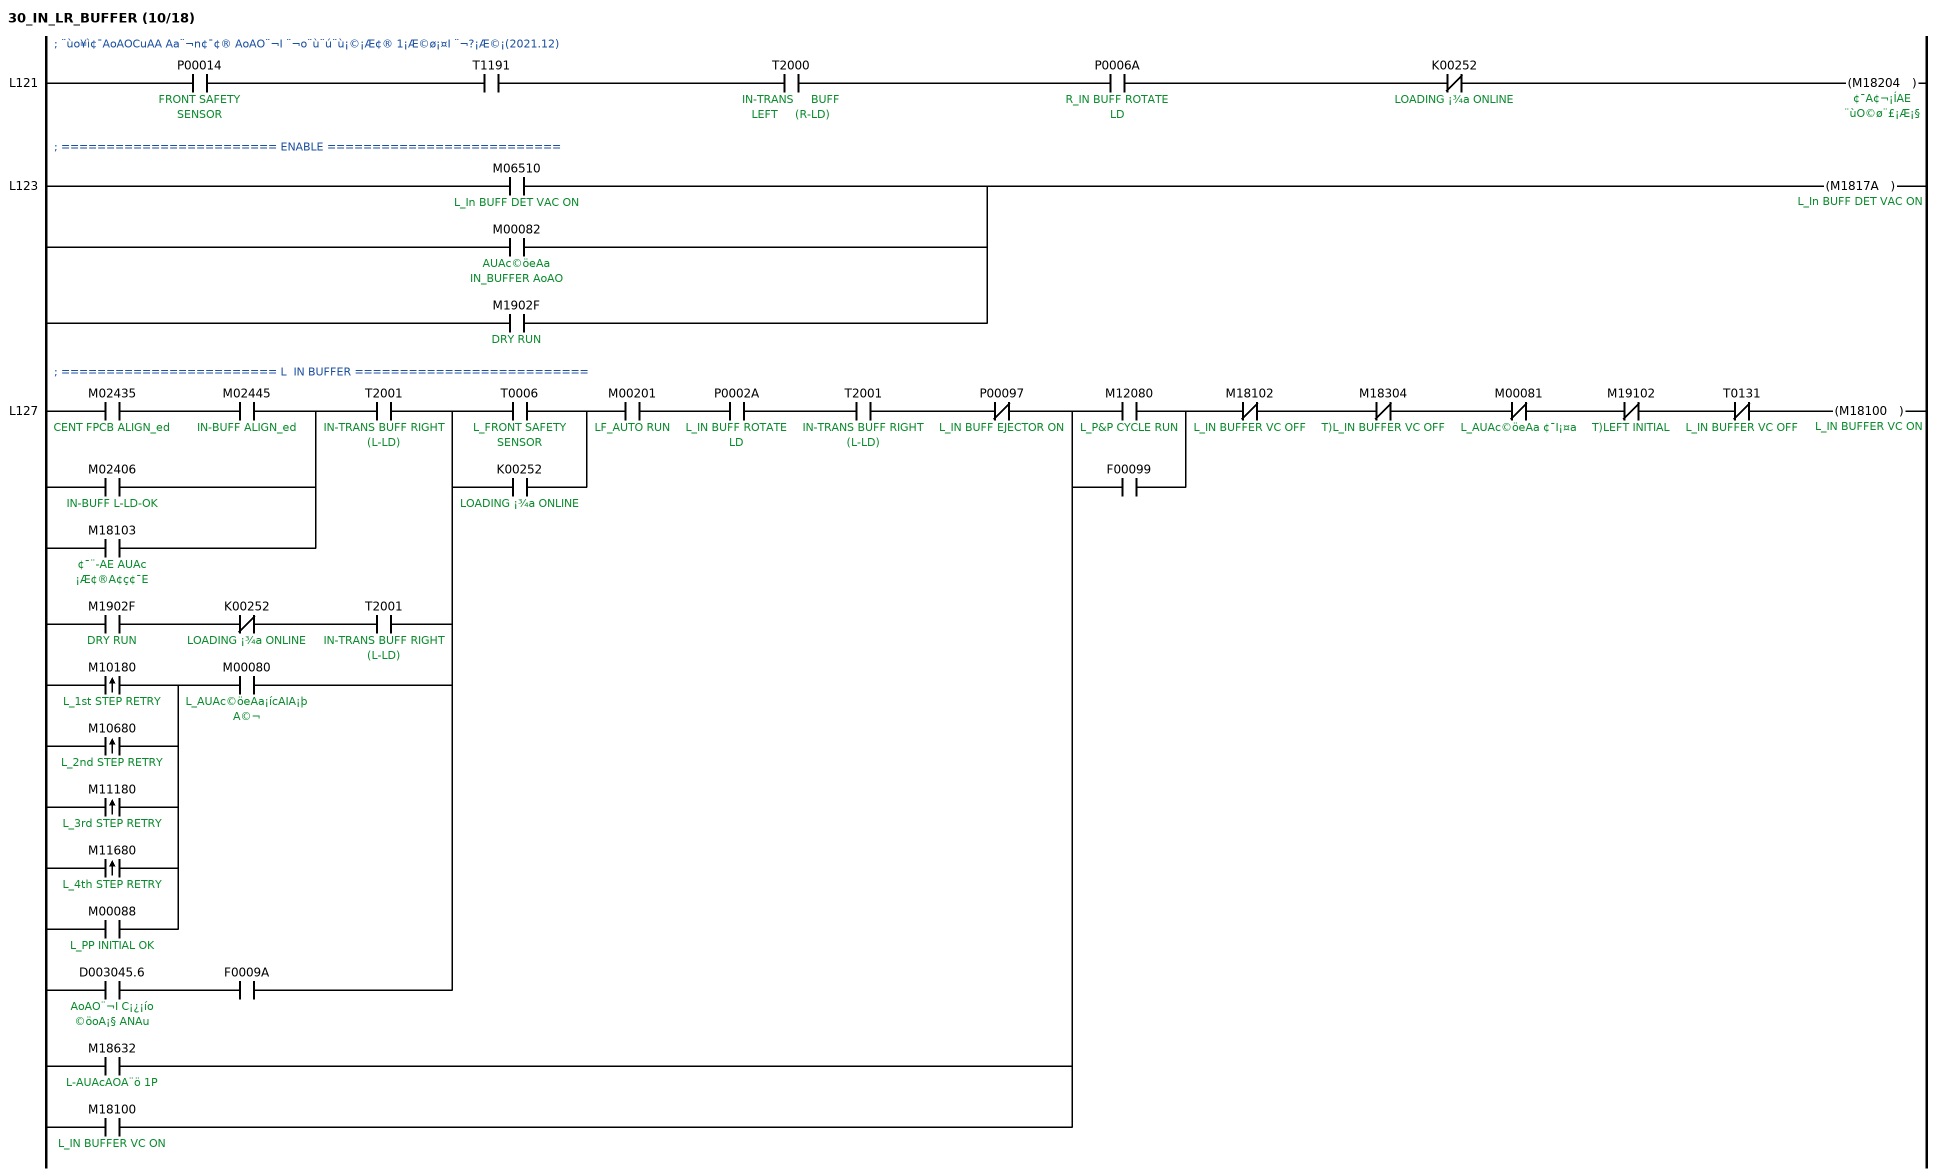
[picture p216: 30_IN_LR_BUFFER rungs L121-L127]
; L121
LOAD      P00014	// FRONT SAFETY SENSOR
AND       T1191
AND       T2000	// IN-TRANS     BUFF     LEFT     (R-LD)
AND       P0006A	// R_IN BUFF ROTATE      LD
AND NOT   K00252	// LOADING ¡¾a ONLINE
OUT       M18204	// ¢¯A¢¬¡ÍAE ¨ùO©ø¨£¡Æ¡§
// output comment: ¨ùo¥ì¢¯AoAOCuAA Aa¨¬n¢¯¢® AoAO¨¬I ¨¬o¨ù¨ú¨ù¡©¡Æ¢® 1¡Æ©ø¡¤I ¨¬?¡Æ©¡(2021.12)
// ======================== ENABLE ==========================
; L123
LOAD      M06510	// L_In BUFF DET VAC ON
OR        M00082	// AUAc©öeAa IN_BUFFER AoAO 
OR        M1902F	// DRY RUN
OUT       M1817A	// L_In BUFF DET VAC ON
// ======================== L  IN BUFFER ==========================
; L127
LOAD      M02435	// CENT FPCB ALIGN_ed
AND       M02445	// IN-BUFF ALIGN_ed
OR        M02406	// IN-BUFF L-LD-OK
OR        M18103	// ¢¯¨­AE AUAc ¡Æ¢®A¢ç¢¯E
AND       T2001	// IN-TRANS BUFF RIGHT     (L-LD)
LOAD      M1902F	// DRY RUN
AND NOT   K00252	// LOADING ¡¾a ONLINE
AND       T2001	// IN-TRANS BUFF RIGHT     (L-LD)
OR LOAD
LOADP     M10180	// L_1st STEP RETRY
ORP       M10680	// L_2nd STEP RETRY
ORP       M11180	// L_3rd STEP RETRY
ORP       M11680	// L_4th STEP RETRY
OR        M00088	// L_PP INITIAL OK
AND       M00080	// L_AUAc©öeAa¡ícAIA¡þA©¬
OR LOAD
LOAD      D003045.6	// AoAO¨¬I C¡¿¡ío ©öoA¡§ ANAu
AND       F0009A
OR LOAD
LOAD      T0006	// L_FRONT SAFETY SENSOR
OR        K00252	// LOADING ¡¾a ONLINE
AND LOAD
AND       M00201	// LF_AUTO RUN
AND       P0002A	// L_IN BUFF ROTATE     LD
AND       T2001	// IN-TRANS BUFF RIGHT     (L-LD)
AND NOT   P00097	// L_IN BUFF EJECTOR ON
OR        M18632	// L-AUAcAOA¨ö 1P
OR        M18100	// L_IN BUFFER VC ON
LOAD      M12080	// L_P&P CYCLE RUN
OR        F00099
AND LOAD
AND NOT   M18102	// L_IN BUFFER VC OFF
AND NOT   M18304	// T)L_IN BUFFER VC OFF
AND NOT   M00081	// L_AUAc©öeAa ¢¯I¡¤a
AND NOT   M19102	// T)LEFT INITIAL
AND NOT   T0131	// L_IN BUFFER VC OFF
OUT       M18100	// L_IN BUFFER VC ON

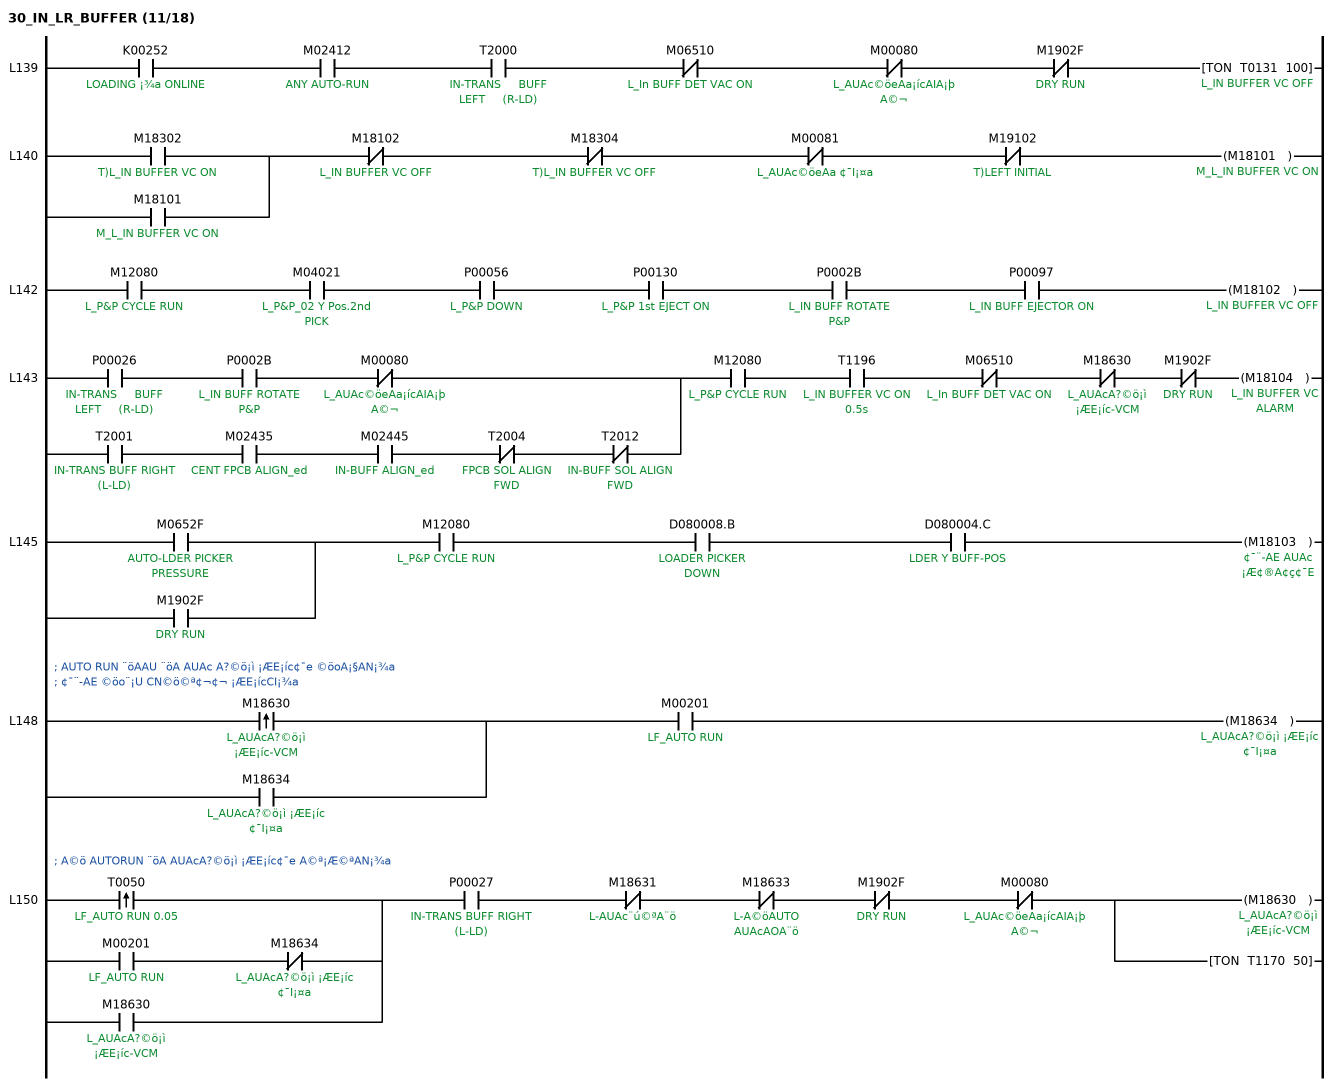
; L139
LOAD      K00252	// LOADING ¡¾a ONLINE
AND       M02412	// ANY AUTO-RUN
AND       T2000	// IN-TRANS     BUFF     LEFT     (R-LD)
AND NOT   M06510	// L_In BUFF DET VAC ON
AND NOT   M00080	// L_AUAc©öeAa¡ícAIA¡þA©¬
AND NOT   M1902F	// DRY RUN
TON       T0131 100	// L_IN BUFFER VC OFF
; L140
LOAD      M18302	// T)L_IN BUFFER VC ON
OR        M18101	// M_L_IN BUFFER VC ON
AND NOT   M18102	// L_IN BUFFER VC OFF
AND NOT   M18304	// T)L_IN BUFFER VC OFF
AND NOT   M00081	// L_AUAc©öeAa ¢¯I¡¤a
AND NOT   M19102	// T)LEFT INITIAL
OUT       M18101	// M_L_IN BUFFER VC ON
; L142
LOAD      M12080	// L_P&P CYCLE RUN
AND       M04021	// L_P&P_02 Y Pos.2nd PICK
AND       P00056	// L_P&P DOWN
AND       P00130	// L_P&P 1st EJECT ON
AND       P0002B	// L_IN BUFF ROTATE      P&P
AND       P00097	// L_IN BUFF EJECTOR ON
OUT       M18102	// L_IN BUFFER VC OFF
; L143
LOAD      P00026	// IN-TRANS     BUFF     LEFT     (R-LD)
AND       P0002B	// L_IN BUFF ROTATE      P&P
AND NOT   M00080	// L_AUAc©öeAa¡ícAIA¡þA©¬
LOAD      T2001	// IN-TRANS BUFF RIGHT     (L-LD)
AND       M02435	// CENT FPCB ALIGN_ed
AND       M02445	// IN-BUFF ALIGN_ed
AND NOT   T2004	// FPCB SOL ALIGN         FWD
AND NOT   T2012	// IN-BUFF SOL ALIGN FWD
OR LOAD
AND       M12080	// L_P&P CYCLE RUN
AND       T1196	// L_IN BUFFER VC ON 0.5s
AND NOT   M06510	// L_In BUFF DET VAC ON
AND NOT   M18630	// L_AUAcA?©ö¡ì ¡ÆE¡íc-VCM
AND NOT   M1902F	// DRY RUN
OUT       M18104	// L_IN BUFFER VC ALARM
; L145
LOAD      M0652F	// AUTO-LDER PICKER PRESSURE
OR        M1902F	// DRY RUN
AND       M12080	// L_P&P CYCLE RUN
AND       D080008.B	// LOADER PICKER DOWN
AND       D080004.C	// LDER Y BUFF-POS
OUT       M18103	// ¢¯¨­AE AUAc ¡Æ¢®A¢ç¢¯E
// AUTO RUN ¨öAAU ¨öA AUAc A?©ö¡ì ¡ÆE¡íc¢¯e ©öoA¡§AN¡¾a
; L148
LOADP     M18630	// L_AUAcA?©ö¡ì ¡ÆE¡íc-VCM
OR        M18634	// L_AUAcA?©ö¡ì ¡ÆE¡íc ¢¯I¡¤a
AND       M00201	// LF_AUTO RUN
OUT       M18634	// L_AUAcA?©ö¡ì ¡ÆE¡íc ¢¯I¡¤a
// output comment: ¢¯¨­AE ©öo¨¡U CN©ö©ª¢¬¢¬ ¡ÆE¡ícCI¡¾a
; L150
LOADP     T0050	// LF_AUTO RUN 0.05
LOAD      M00201	// LF_AUTO RUN
AND NOT   M18634	// L_AUAcA?©ö¡ì ¡ÆE¡íc ¢¯I¡¤a
OR LOAD
OR        M18630	// L_AUAcA?©ö¡ì ¡ÆE¡íc-VCM
AND       P00027	// IN-TRANS BUFF RIGHT     (L-LD)
AND NOT   M18631	// L-AUAc¨ú©ªA¨ö
AND NOT   M18633	// L-A©öAUTO AUAcAOA¨ö
AND NOT   M1902F	// DRY RUN
AND NOT   M00080	// L_AUAc©öeAa¡ícAIA¡þA©¬
OUT       M18630	// L_AUAcA?©ö¡ì ¡ÆE¡íc-VCM
TON       T1170 50
// output comment: A©ö AUTORUN ¨öA AUAcA?©ö¡ì ¡ÆE¡íc¢¯e A©ª¡Æ©ªAN¡¾a

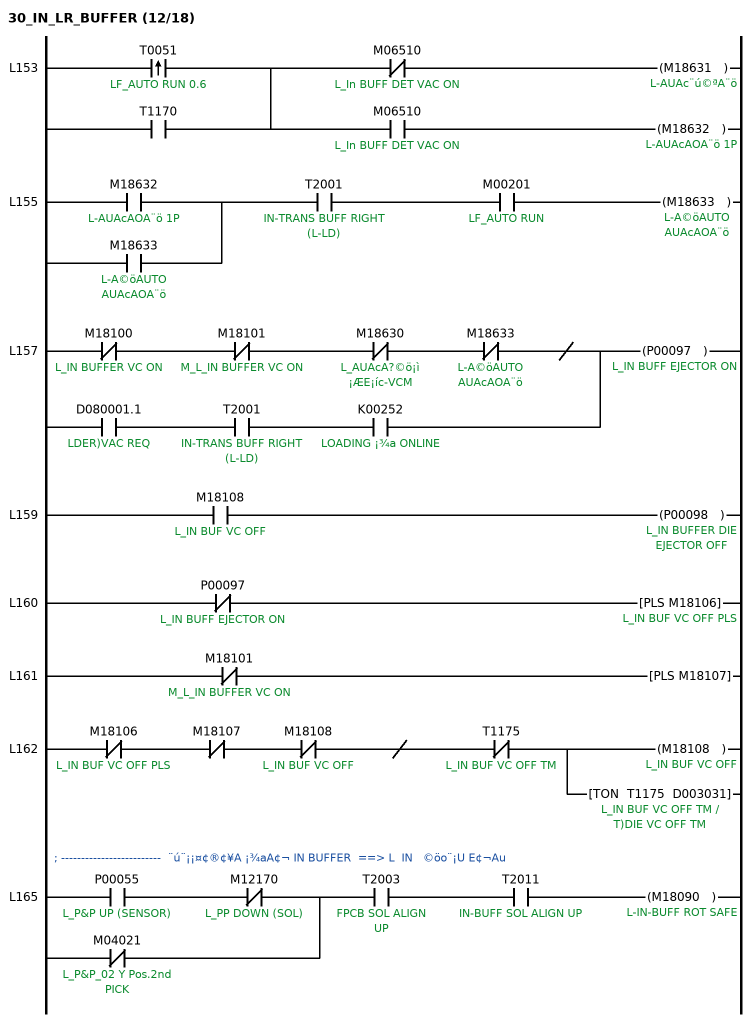
; L153
LOADP     T0051	// LF_AUTO RUN 0.6
OR        T1170
MPUSH
AND NOT   M06510	// L_In BUFF DET VAC ON
OUT       M18631	// L-AUAc¨ú©ªA¨ö
MPOP
AND       M06510	// L_In BUFF DET VAC ON
OUT       M18632	// L-AUAcAOA¨ö 1P
; L155
LOAD      M18632	// L-AUAcAOA¨ö 1P
OR        M18633	// L-A©öAUTO AUAcAOA¨ö
AND       T2001	// IN-TRANS BUFF RIGHT     (L-LD)
AND       M00201	// LF_AUTO RUN
OUT       M18633	// L-A©öAUTO AUAcAOA¨ö
; L157
LOAD NOT  M18100	// L_IN BUFFER VC ON
AND NOT   M18101	// M_L_IN BUFFER VC ON
AND NOT   M18630	// L_AUAcA?©ö¡ì ¡ÆE¡íc-VCM
AND NOT   M18633	// L-A©öAUTO AUAcAOA¨ö
NOT
LOAD      D080001.1	// LDER)VAC REQ
AND       T2001	// IN-TRANS BUFF RIGHT     (L-LD)
AND       K00252	// LOADING ¡¾a ONLINE
OR LOAD
OUT       P00097	// L_IN BUFF EJECTOR ON
; L159
LOAD      M18108	// L_IN BUF VC OFF
OUT       P00098	// L_IN BUFFER DIE EJECTOR OFF
; L160
LOAD NOT  P00097	// L_IN BUFF EJECTOR ON
OUTP      M18106	// L_IN BUF VC OFF PLS
; L161
LOAD NOT  M18101	// M_L_IN BUFFER VC ON
OUTP      M18107
; L162
LOAD NOT  M18106	// L_IN BUF VC OFF PLS
AND NOT   M18107
AND NOT   M18108	// L_IN BUF VC OFF
NOT
AND NOT   T1175	// L_IN BUF VC OFF TM
OUT       M18108	// L_IN BUF VC OFF
TON       T1175 D003031	// L_IN BUF VC OFF TM / T)DIE VC OFF TM
// -------------------------  ¨ú¨¡¡¤¢®¢¥A ¡¾aA¢¬ IN BUFFER  ==> L  IN   ©öo¨¡U E¢¬Au
; L165
LOAD      P00055	// L_P&P UP (SENSOR)
AND NOT   M12170	// L_PP DOWN (SOL)
OR NOT    M04021	// L_P&P_02 Y Pos.2nd PICK
AND       T2003	// FPCB SOL ALIGN         UP
AND       T2011	// IN-BUFF SOL ALIGN UP
OUT       M18090	// L-IN-BUFF ROT SAFE

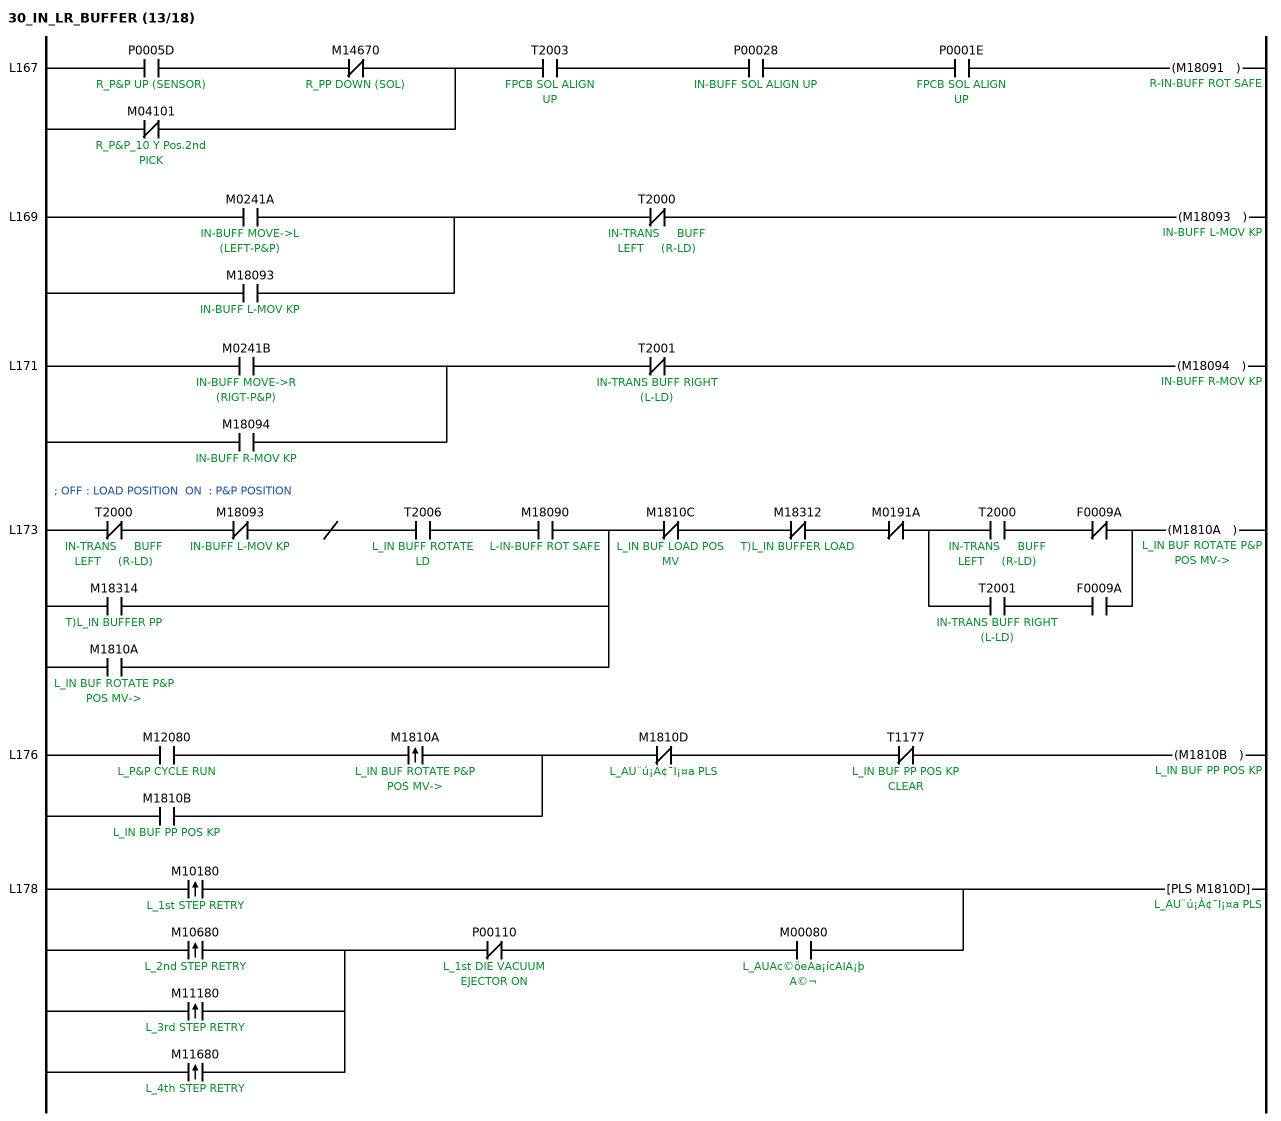
; L167
LOAD      P0005D	// R_P&P UP (SENSOR)
AND NOT   M14670	// R_PP DOWN (SOL)
OR NOT    M04101	// R_P&P_10 Y Pos.2nd PICK
AND       T2003	// FPCB SOL ALIGN         UP
AND       P00028	// IN-BUFF SOL ALIGN UP
AND       P0001E	// FPCB SOL ALIGN         UP
OUT       M18091	// R-IN-BUFF ROT SAFE
; L169
LOAD      M0241A	// IN-BUFF MOVE->L (LEFT-P&P)
OR        M18093	// IN-BUFF L-MOV KP
AND NOT   T2000	// IN-TRANS     BUFF     LEFT     (R-LD)
OUT       M18093	// IN-BUFF L-MOV KP
; L171
LOAD      M0241B	// IN-BUFF MOVE->R (RIGT-P&P)
OR        M18094	// IN-BUFF R-MOV KP
AND NOT   T2001	// IN-TRANS BUFF RIGHT     (L-LD)
OUT       M18094	// IN-BUFF R-MOV KP
; L173
LOAD NOT  T2000	// IN-TRANS     BUFF     LEFT     (R-LD)
AND NOT   M18093	// IN-BUFF L-MOV KP
NOT
AND       T2006	// L_IN BUFF ROTATE     LD
AND       M18090	// L-IN-BUFF ROT SAFE
OR        M18314	// T)L_IN BUFFER PP
OR        M1810A	// L_IN BUF ROTATE P&P POS MV->
AND NOT   M1810C	// L_IN BUF LOAD POS MV
AND NOT   M18312	// T)L_IN BUFFER LOAD
AND NOT   M0191A
LOAD      T2000	// IN-TRANS     BUFF     LEFT     (R-LD)
AND NOT   F0009A
LOAD      T2001	// IN-TRANS BUFF RIGHT     (L-LD)
AND       F0009A
OR LOAD
AND LOAD
OUT       M1810A	// L_IN BUF ROTATE P&P POS MV->
// output comment: OFF : LOAD POSITION  ON  : P&P POSITION
; L176
LOAD      M12080	// L_P&P CYCLE RUN
ANDP      M1810A	// L_IN BUF ROTATE P&P POS MV->
OR        M1810B	// L_IN BUF PP POS KP
AND NOT   M1810D	// L_AU¨ú¡À¢¯I¡¤a PLS
AND NOT   T1177	// L_IN BUF PP POS KP CLEAR
OUT       M1810B	// L_IN BUF PP POS KP
; L178
LOADP     M10180	// L_1st STEP RETRY
LOADP     M10680	// L_2nd STEP RETRY
ORP       M11180	// L_3rd STEP RETRY
ORP       M11680	// L_4th STEP RETRY
AND NOT   P00110	// L_1st DIE VACUUM EJECTOR ON
AND       M00080	// L_AUAc©öeAa¡ícAIA¡þA©¬
OR LOAD
OUTP      M1810D	// L_AU¨ú¡À¢¯I¡¤a PLS

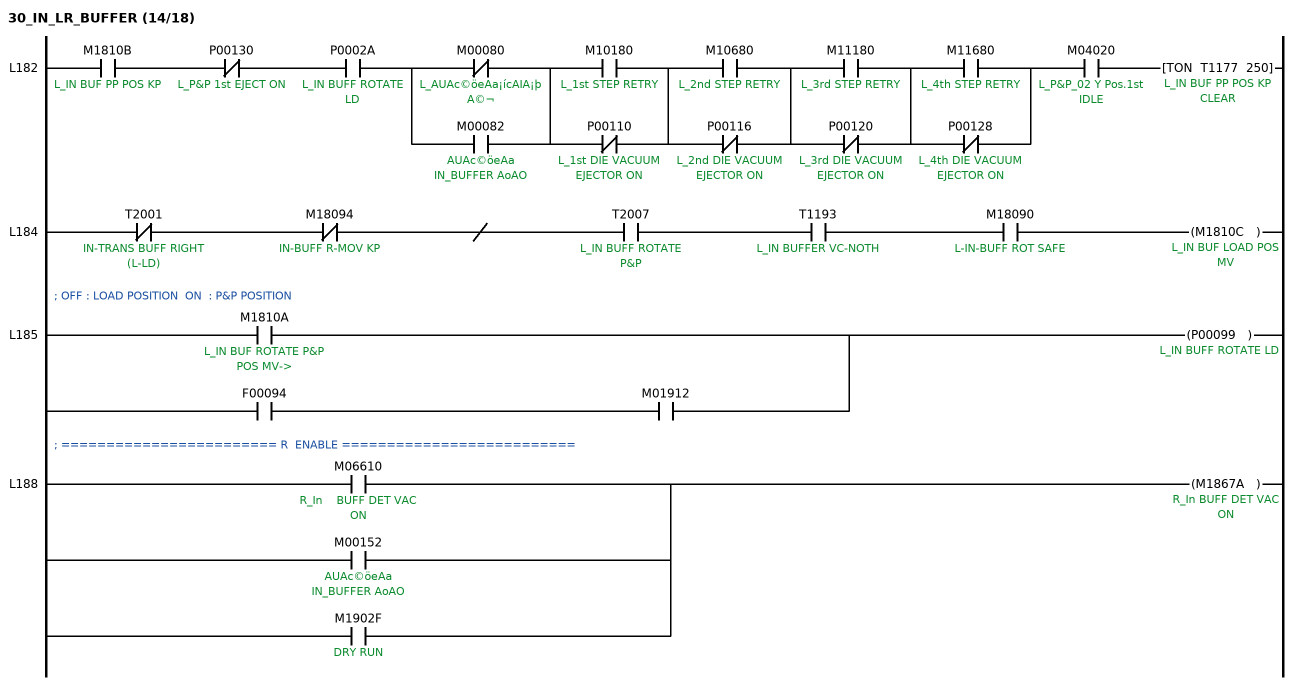
; L182
LOAD      M1810B	// L_IN BUF PP POS KP
AND NOT   P00130	// L_P&P 1st EJECT ON
AND       P0002A	// L_IN BUFF ROTATE     LD
LOAD NOT  M00080	// L_AUAc©öeAa¡ícAIA¡þA©¬
OR        M00082	// AUAc©öeAa IN_BUFFER AoAO 
AND LOAD
LOAD      M10180	// L_1st STEP RETRY
OR NOT    P00110	// L_1st DIE VACUUM EJECTOR ON
AND LOAD
LOAD      M10680	// L_2nd STEP RETRY
OR NOT    P00116	// L_2nd DIE VACUUM EJECTOR ON
AND LOAD
LOAD      M11180	// L_3rd STEP RETRY
OR NOT    P00120	// L_3rd DIE VACUUM EJECTOR ON
AND LOAD
LOAD      M11680	// L_4th STEP RETRY
OR NOT    P00128	// L_4th DIE VACUUM EJECTOR ON
AND LOAD
AND       M04020	// L_P&P_02 Y Pos.1st IDLE
TON       T1177 250	// L_IN BUF PP POS KP CLEAR
; L184
LOAD NOT  T2001	// IN-TRANS BUFF RIGHT     (L-LD)
AND NOT   M18094	// IN-BUFF R-MOV KP
NOT
AND       T2007	// L_IN BUFF ROTATE      P&P
AND       T1193	// L_IN BUFFER VC-NOTH
AND       M18090	// L-IN-BUFF ROT SAFE
OUT       M1810C	// L_IN BUF LOAD POS MV
; L185
LOAD      M1810A	// L_IN BUF ROTATE P&P POS MV->
LOAD      F00094
AND       M01912
OR LOAD
OUT       P00099	// L_IN BUFF ROTATE LD
// output comment: OFF : LOAD POSITION  ON  : P&P POSITION
// ======================== R  ENABLE ==========================
; L188
LOAD      M06610	// R_In    BUFF DET VAC ON
OR        M00152	// AUAc©öeAa IN_BUFFER AoAO 
OR        M1902F	// DRY RUN
OUT       M1867A	// R_In BUFF DET VAC ON

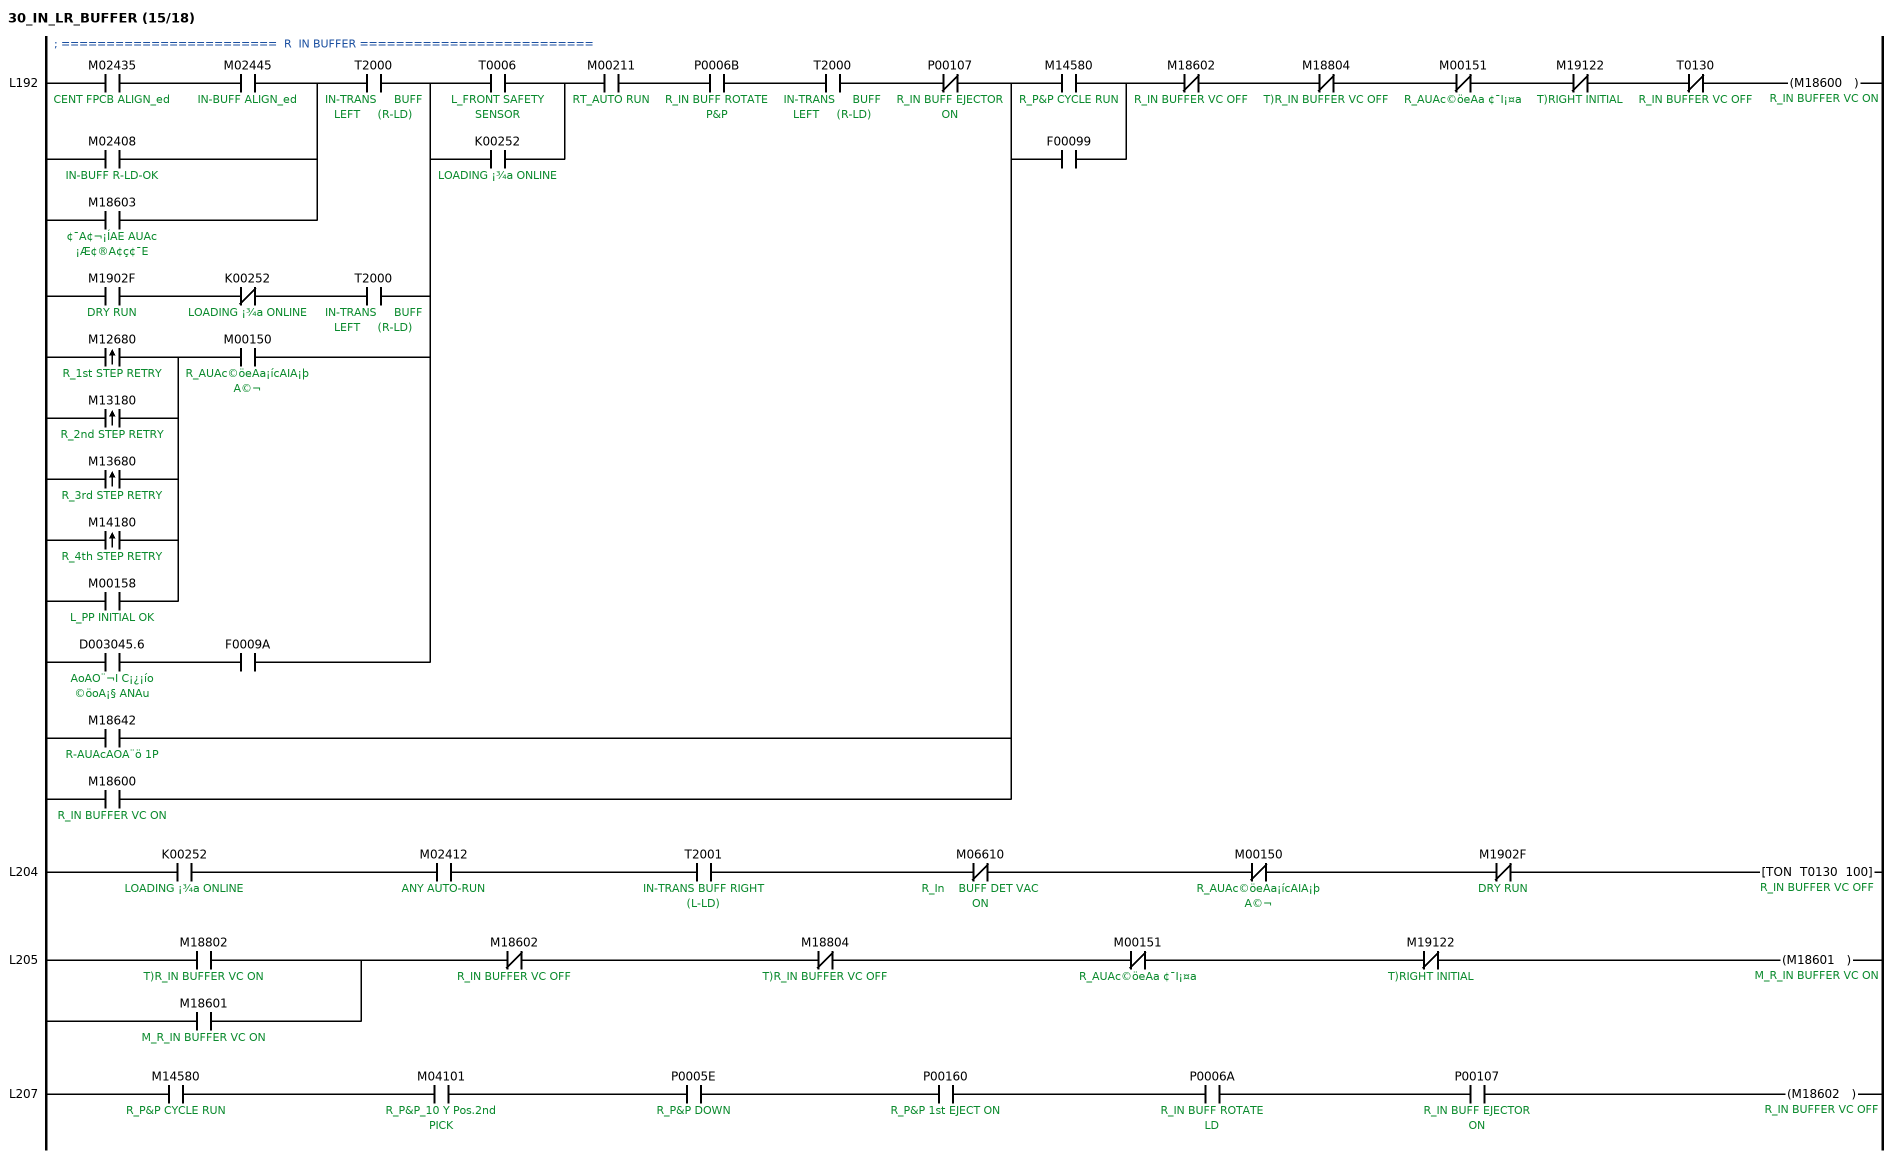
// ========================  R  IN BUFFER ==========================
; L192
LOAD      M02435	// CENT FPCB ALIGN_ed
AND       M02445	// IN-BUFF ALIGN_ed
OR        M02408	// IN-BUFF R-LD-OK
OR        M18603	// ¢¯A¢¬¡ÍAE AUAc ¡Æ¢®A¢ç¢¯E
AND       T2000	// IN-TRANS     BUFF     LEFT     (R-LD)
LOAD      M1902F	// DRY RUN
AND NOT   K00252	// LOADING ¡¾a ONLINE
AND       T2000	// IN-TRANS     BUFF     LEFT     (R-LD)
OR LOAD
LOADP     M12680	// R_1st STEP RETRY
ORP       M13180	// R_2nd STEP RETRY
ORP       M13680	// R_3rd STEP RETRY
ORP       M14180	// R_4th STEP RETRY
OR        M00158	// L_PP INITIAL OK
AND       M00150	// R_AUAc©öeAa¡ícAIA¡þA©¬
OR LOAD
LOAD      D003045.6	// AoAO¨¬I C¡¿¡ío ©öoA¡§ ANAu
AND       F0009A
OR LOAD
LOAD      T0006	// L_FRONT SAFETY SENSOR
OR        K00252	// LOADING ¡¾a ONLINE
AND LOAD
AND       M00211	// RT_AUTO RUN
AND       P0006B	// R_IN BUFF ROTATE      P&P
AND       T2000	// IN-TRANS     BUFF     LEFT     (R-LD)
AND NOT   P00107	// R_IN BUFF EJECTOR ON
OR        M18642	// R-AUAcAOA¨ö 1P
OR        M18600	// R_IN BUFFER VC ON
LOAD      M14580	// R_P&P CYCLE RUN
OR        F00099
AND LOAD
AND NOT   M18602	// R_IN BUFFER VC OFF
AND NOT   M18804	// T)R_IN BUFFER VC OFF
AND NOT   M00151	// R_AUAc©öeAa ¢¯I¡¤a
AND NOT   M19122	// T)RIGHT INITIAL
AND NOT   T0130	// R_IN BUFFER VC OFF
OUT       M18600	// R_IN BUFFER VC ON
; L204
LOAD      K00252	// LOADING ¡¾a ONLINE
AND       M02412	// ANY AUTO-RUN
AND       T2001	// IN-TRANS BUFF RIGHT     (L-LD)
AND NOT   M06610	// R_In    BUFF DET VAC ON
AND NOT   M00150	// R_AUAc©öeAa¡ícAIA¡þA©¬
AND NOT   M1902F	// DRY RUN
TON       T0130 100	// R_IN BUFFER VC OFF
; L205
LOAD      M18802	// T)R_IN BUFFER VC ON
OR        M18601	// M_R_IN BUFFER VC ON
AND NOT   M18602	// R_IN BUFFER VC OFF
AND NOT   M18804	// T)R_IN BUFFER VC OFF
AND NOT   M00151	// R_AUAc©öeAa ¢¯I¡¤a
AND NOT   M19122	// T)RIGHT INITIAL
OUT       M18601	// M_R_IN BUFFER VC ON
; L207
LOAD      M14580	// R_P&P CYCLE RUN
AND       M04101	// R_P&P_10 Y Pos.2nd PICK
AND       P0005E	// R_P&P DOWN
AND       P00160	// R_P&P 1st EJECT ON
AND       P0006A	// R_IN BUFF ROTATE      LD
AND       P00107	// R_IN BUFF EJECTOR ON
OUT       M18602	// R_IN BUFFER VC OFF

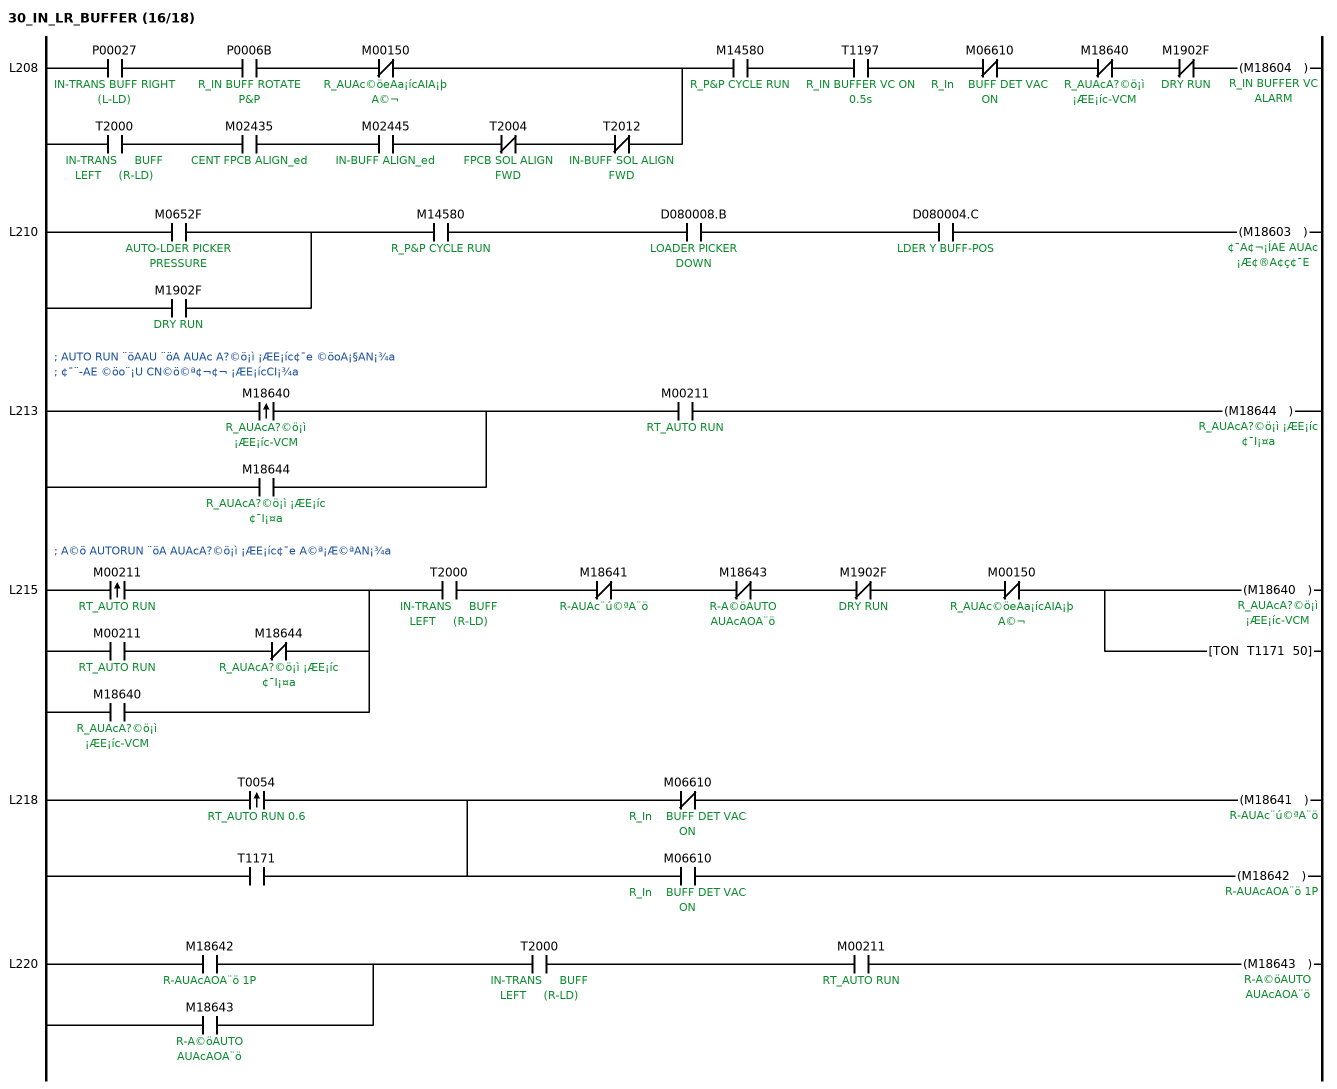
; L208
LOAD      P00027	// IN-TRANS BUFF RIGHT     (L-LD)
AND       P0006B	// R_IN BUFF ROTATE      P&P
AND NOT   M00150	// R_AUAc©öeAa¡ícAIA¡þA©¬
LOAD      T2000	// IN-TRANS     BUFF     LEFT     (R-LD)
AND       M02435	// CENT FPCB ALIGN_ed
AND       M02445	// IN-BUFF ALIGN_ed
AND NOT   T2004	// FPCB SOL ALIGN         FWD
AND NOT   T2012	// IN-BUFF SOL ALIGN FWD
OR LOAD
AND       M14580	// R_P&P CYCLE RUN
AND       T1197	// R_IN BUFFER VC ON 0.5s
AND NOT   M06610	// R_In    BUFF DET VAC ON
AND NOT   M18640	// R_AUAcA?©ö¡ì ¡ÆE¡íc-VCM
AND NOT   M1902F	// DRY RUN
OUT       M18604	// R_IN BUFFER VC ALARM
; L210
LOAD      M0652F	// AUTO-LDER PICKER PRESSURE
OR        M1902F	// DRY RUN
AND       M14580	// R_P&P CYCLE RUN
AND       D080008.B	// LOADER PICKER DOWN
AND       D080004.C	// LDER Y BUFF-POS
OUT       M18603	// ¢¯A¢¬¡ÍAE AUAc ¡Æ¢®A¢ç¢¯E
// AUTO RUN ¨öAAU ¨öA AUAc A?©ö¡ì ¡ÆE¡íc¢¯e ©öoA¡§AN¡¾a
; L213
LOADP     M18640	// R_AUAcA?©ö¡ì ¡ÆE¡íc-VCM
OR        M18644	// R_AUAcA?©ö¡ì ¡ÆE¡íc ¢¯I¡¤a
AND       M00211	// RT_AUTO RUN
OUT       M18644	// R_AUAcA?©ö¡ì ¡ÆE¡íc ¢¯I¡¤a
// output comment: ¢¯¨­AE ©öo¨¡U CN©ö©ª¢¬¢¬ ¡ÆE¡ícCI¡¾a
; L215
LOADP     M00211	// RT_AUTO RUN
LOAD      M00211	// RT_AUTO RUN
AND NOT   M18644	// R_AUAcA?©ö¡ì ¡ÆE¡íc ¢¯I¡¤a
OR LOAD
OR        M18640	// R_AUAcA?©ö¡ì ¡ÆE¡íc-VCM
AND       T2000	// IN-TRANS     BUFF     LEFT     (R-LD)
AND NOT   M18641	// R-AUAc¨ú©ªA¨ö
AND NOT   M18643	// R-A©öAUTO AUAcAOA¨ö
AND NOT   M1902F	// DRY RUN
AND NOT   M00150	// R_AUAc©öeAa¡ícAIA¡þA©¬
OUT       M18640	// R_AUAcA?©ö¡ì ¡ÆE¡íc-VCM
TON       T1171 50
// output comment: A©ö AUTORUN ¨öA AUAcA?©ö¡ì ¡ÆE¡íc¢¯e A©ª¡Æ©ªAN¡¾a
; L218
LOADP     T0054	// RT_AUTO RUN 0.6
OR        T1171
MPUSH
AND NOT   M06610	// R_In    BUFF DET VAC ON
OUT       M18641	// R-AUAc¨ú©ªA¨ö
MPOP
AND       M06610	// R_In    BUFF DET VAC ON
OUT       M18642	// R-AUAcAOA¨ö 1P
; L220
LOAD      M18642	// R-AUAcAOA¨ö 1P
OR        M18643	// R-A©öAUTO AUAcAOA¨ö
AND       T2000	// IN-TRANS     BUFF     LEFT     (R-LD)
AND       M00211	// RT_AUTO RUN
OUT       M18643	// R-A©öAUTO AUAcAOA¨ö

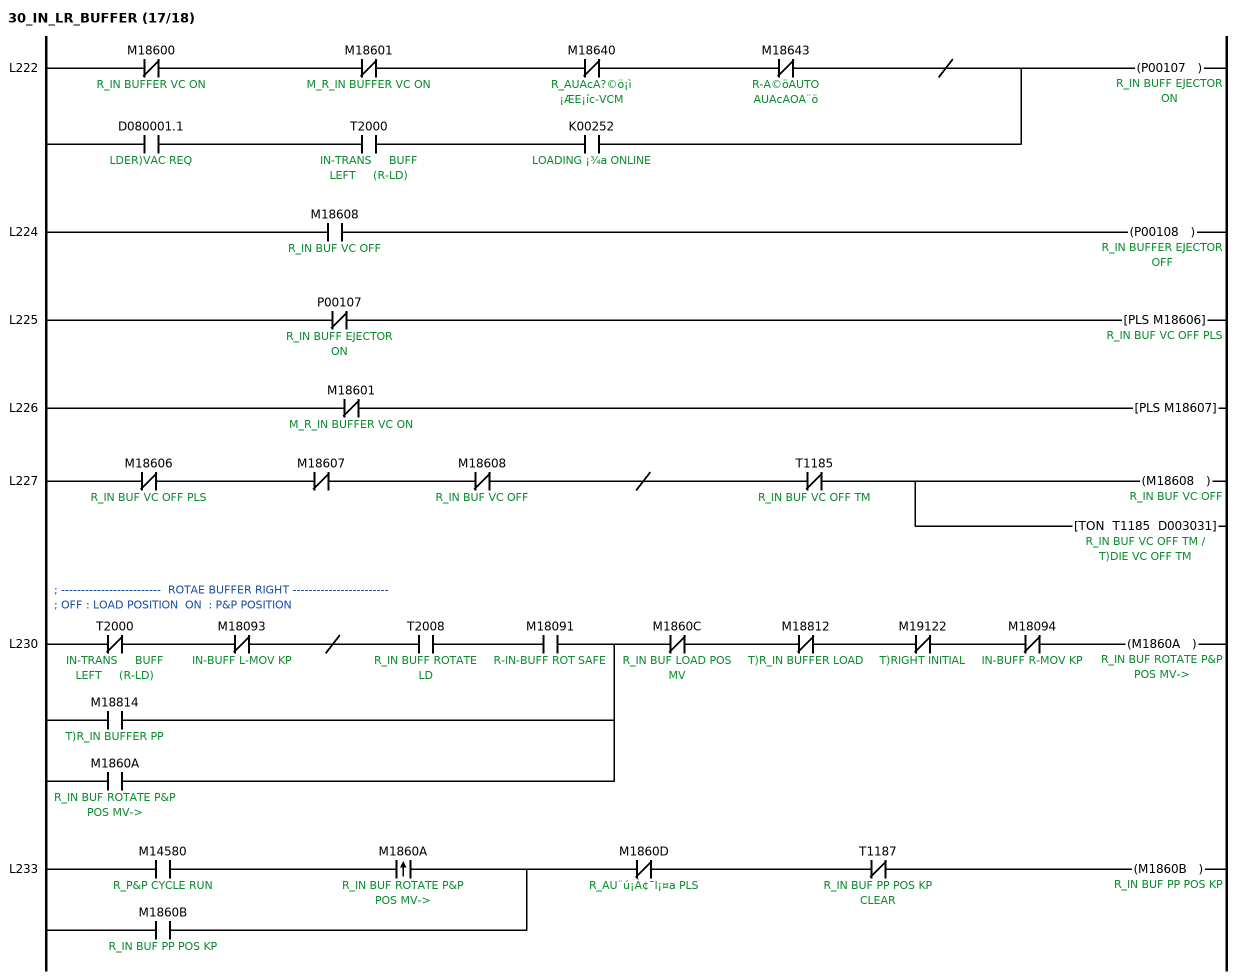
; L222
LOAD NOT  M18600	// R_IN BUFFER VC ON
AND NOT   M18601	// M_R_IN BUFFER VC ON
AND NOT   M18640	// R_AUAcA?©ö¡ì ¡ÆE¡íc-VCM
AND NOT   M18643	// R-A©öAUTO AUAcAOA¨ö
NOT
LOAD      D080001.1	// LDER)VAC REQ
AND       T2000	// IN-TRANS     BUFF     LEFT     (R-LD)
AND       K00252	// LOADING ¡¾a ONLINE
OR LOAD
OUT       P00107	// R_IN BUFF EJECTOR ON
; L224
LOAD      M18608	// R_IN BUF VC OFF
OUT       P00108	// R_IN BUFFER EJECTOR OFF
; L225
LOAD NOT  P00107	// R_IN BUFF EJECTOR ON
OUTP      M18606	// R_IN BUF VC OFF PLS
; L226
LOAD NOT  M18601	// M_R_IN BUFFER VC ON
OUTP      M18607
; L227
LOAD NOT  M18606	// R_IN BUF VC OFF PLS
AND NOT   M18607
AND NOT   M18608	// R_IN BUF VC OFF
NOT
AND NOT   T1185	// R_IN BUF VC OFF TM
OUT       M18608	// R_IN BUF VC OFF
TON       T1185 D003031	// R_IN BUF VC OFF TM / T)DIE VC OFF TM
// -------------------------  ROTAE BUFFER RIGHT ------------------------
; L230
LOAD NOT  T2000	// IN-TRANS     BUFF     LEFT     (R-LD)
AND NOT   M18093	// IN-BUFF L-MOV KP
NOT
AND       T2008	// R_IN BUFF ROTATE      LD
AND       M18091	// R-IN-BUFF ROT SAFE
OR        M18814	// T)R_IN BUFFER PP
OR        M1860A	// R_IN BUF ROTATE P&P POS MV->
AND NOT   M1860C	// R_IN BUF LOAD POS MV
AND NOT   M18812	// T)R_IN BUFFER LOAD
AND NOT   M19122	// T)RIGHT INITIAL
AND NOT   M18094	// IN-BUFF R-MOV KP
OUT       M1860A	// R_IN BUF ROTATE P&P POS MV->
// output comment: OFF : LOAD POSITION  ON  : P&P POSITION
; L233
LOAD      M14580	// R_P&P CYCLE RUN
ANDP      M1860A	// R_IN BUF ROTATE P&P POS MV->
OR        M1860B	// R_IN BUF PP POS KP
AND NOT   M1860D	// R_AU¨ú¡À¢¯I¡¤a PLS
AND NOT   T1187	// R_IN BUF PP POS KP CLEAR
OUT       M1860B	// R_IN BUF PP POS KP

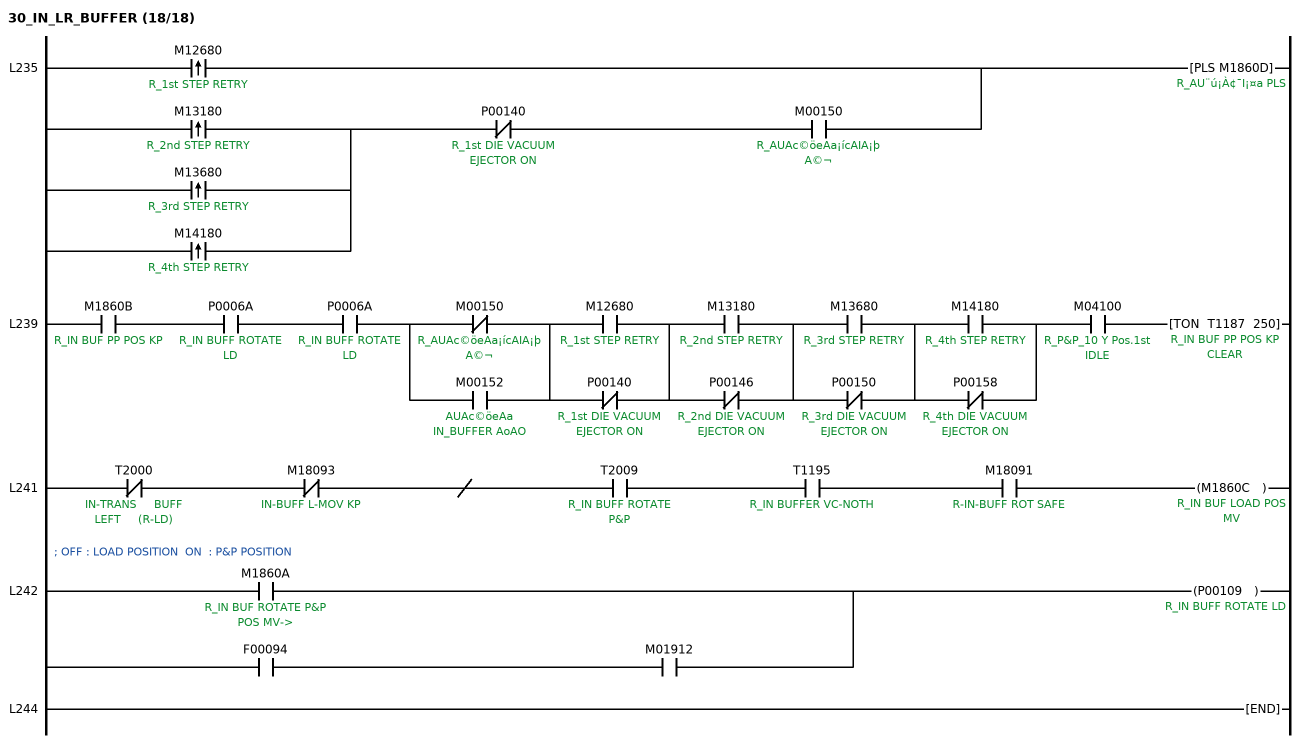
; L235
LOADP     M12680	// R_1st STEP RETRY
LOADP     M13180	// R_2nd STEP RETRY
ORP       M13680	// R_3rd STEP RETRY
ORP       M14180	// R_4th STEP RETRY
AND NOT   P00140	// R_1st DIE VACUUM EJECTOR ON
AND       M00150	// R_AUAc©öeAa¡ícAIA¡þA©¬
OR LOAD
OUTP      M1860D	// R_AU¨ú¡À¢¯I¡¤a PLS
; L239
LOAD      M1860B	// R_IN BUF PP POS KP
AND       P0006A	// R_IN BUFF ROTATE      LD
AND       P0006A	// R_IN BUFF ROTATE      LD
LOAD NOT  M00150	// R_AUAc©öeAa¡ícAIA¡þA©¬
OR        M00152	// AUAc©öeAa IN_BUFFER AoAO 
AND LOAD
LOAD      M12680	// R_1st STEP RETRY
OR NOT    P00140	// R_1st DIE VACUUM EJECTOR ON
AND LOAD
LOAD      M13180	// R_2nd STEP RETRY
OR NOT    P00146	// R_2nd DIE VACUUM EJECTOR ON
AND LOAD
LOAD      M13680	// R_3rd STEP RETRY
OR NOT    P00150	// R_3rd DIE VACUUM EJECTOR ON
AND LOAD
LOAD      M14180	// R_4th STEP RETRY
OR NOT    P00158	// R_4th DIE VACUUM EJECTOR ON
AND LOAD
AND       M04100	// R_P&P_10 Y Pos.1st IDLE
TON       T1187 250	// R_IN BUF PP POS KP CLEAR
; L241
LOAD NOT  T2000	// IN-TRANS     BUFF     LEFT     (R-LD)
AND NOT   M18093	// IN-BUFF L-MOV KP
NOT
AND       T2009	// R_IN BUFF ROTATE      P&P
AND       T1195	// R_IN BUFFER VC-NOTH
AND       M18091	// R-IN-BUFF ROT SAFE
OUT       M1860C	// R_IN BUF LOAD POS MV
; L242
LOAD      M1860A	// R_IN BUF ROTATE P&P POS MV->
LOAD      F00094
AND       M01912
OR LOAD
OUT       P00109	// R_IN BUFF ROTATE LD
// output comment: OFF : LOAD POSITION  ON  : P&P POSITION
; L244
END

PROGRAM 31_OUT_LR_BUFFER (task: ¨ö¨¬A¥ì CA¡¤I¡¾¡¿¡¤¡Í)

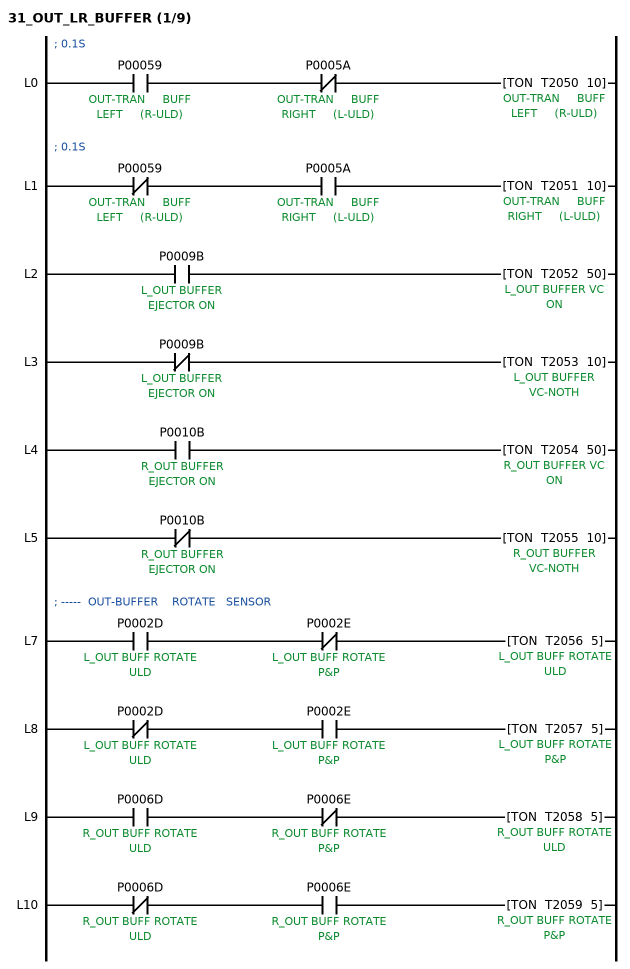
; L0
LOAD      P00059	// OUT-TRAN     BUFF     LEFT     (R-ULD)
AND NOT   P0005A	// OUT-TRAN     BUFF     RIGHT     (L-ULD)
TON       T2050 10	// OUT-TRAN     BUFF     LEFT     (R-ULD)
// output comment: 0.1S
; L1
LOAD NOT  P00059	// OUT-TRAN     BUFF     LEFT     (R-ULD)
AND       P0005A	// OUT-TRAN     BUFF     RIGHT     (L-ULD)
TON       T2051 10	// OUT-TRAN     BUFF     RIGHT     (L-ULD)
// output comment: 0.1S
; L2
LOAD      P0009B	// L_OUT BUFFER EJECTOR ON
TON       T2052 50	// L_OUT BUFFER VC ON
; L3
LOAD NOT  P0009B	// L_OUT BUFFER EJECTOR ON
TON       T2053 10	// L_OUT BUFFER VC-NOTH
; L4
LOAD      P0010B	// R_OUT BUFFER EJECTOR ON
TON       T2054 50	// R_OUT BUFFER VC ON
; L5
LOAD NOT  P0010B	// R_OUT BUFFER EJECTOR ON
TON       T2055 10	// R_OUT BUFFER VC-NOTH
// -----  OUT-BUFFER    ROTATE   SENSOR
; L7
LOAD      P0002D	// L_OUT BUFF ROTATE     ULD
AND NOT   P0002E	// L_OUT BUFF ROTATE      P&P
TON       T2056 5	// L_OUT BUFF ROTATE     ULD
; L8
LOAD NOT  P0002D	// L_OUT BUFF ROTATE     ULD
AND       P0002E	// L_OUT BUFF ROTATE      P&P
TON       T2057 5	// L_OUT BUFF ROTATE      P&P
; L9
LOAD      P0006D	// R_OUT BUFF ROTATE      ULD
AND NOT   P0006E	// R_OUT BUFF ROTATE      P&P
TON       T2058 5	// R_OUT BUFF ROTATE      ULD
; L10
LOAD NOT  P0006D	// R_OUT BUFF ROTATE      ULD
AND       P0006E	// R_OUT BUFF ROTATE      P&P
TON       T2059 5	// R_OUT BUFF ROTATE      P&P

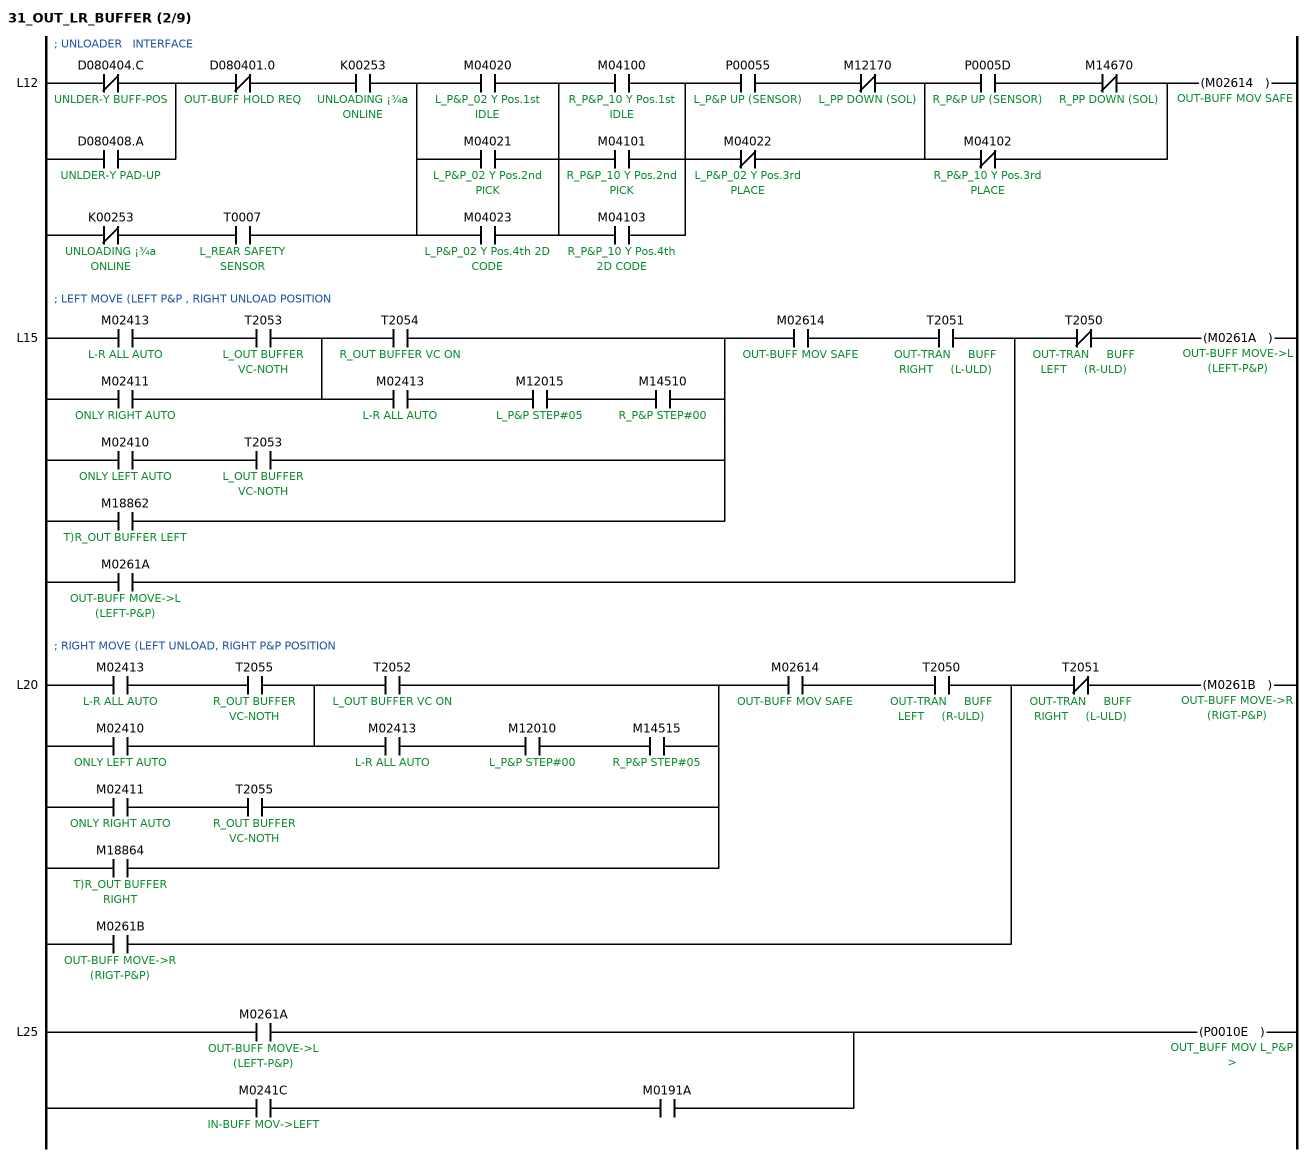
//  UNLOADER   INTERFACE
; L12
LOAD NOT  D080404.C	// UNLDER-Y BUFF-POS
OR        D080408.A	// UNLDER-Y PAD-UP
AND NOT   D080401.0	// OUT-BUFF HOLD REQ
AND       K00253	// UNLOADING ¡¾a ONLINE
LOAD NOT  K00253	// UNLOADING ¡¾a ONLINE
AND       T0007	// L_REAR SAFETY SENSOR
OR LOAD
LOAD      M04020	// L_P&P_02 Y Pos.1st IDLE
OR        M04021	// L_P&P_02 Y Pos.2nd PICK
OR        M04023	// L_P&P_02 Y Pos.4th 2D CODE
AND LOAD
LOAD      M04100	// R_P&P_10 Y Pos.1st IDLE
OR        M04101	// R_P&P_10 Y Pos.2nd PICK
OR        M04103	// R_P&P_10 Y Pos.4th 2D CODE
AND LOAD
LOAD      P00055	// L_P&P UP (SENSOR)
AND NOT   M12170	// L_PP DOWN (SOL)
OR NOT    M04022	// L_P&P_02 Y Pos.3rd PLACE
AND LOAD
LOAD      P0005D	// R_P&P UP (SENSOR)
AND NOT   M14670	// R_PP DOWN (SOL)
OR NOT    M04102	// R_P&P_10 Y Pos.3rd PLACE
AND LOAD
OUT       M02614	// OUT-BUFF MOV SAFE
; L15
LOAD      M02413	// L-R ALL AUTO
AND       T2053	// L_OUT BUFFER VC-NOTH
OR        M02411	// ONLY RIGHT AUTO
LOAD      T2054	// R_OUT BUFFER VC ON
LOAD      M02413	// L-R ALL AUTO
AND       M12015	// L_P&P STEP#05
AND       M14510	// R_P&P STEP#00
OR LOAD
AND LOAD
LOAD      M02410	// ONLY LEFT AUTO
AND       T2053	// L_OUT BUFFER VC-NOTH
OR LOAD
OR        M18862	// T)R_OUT BUFFER LEFT
AND       M02614	// OUT-BUFF MOV SAFE
AND       T2051	// OUT-TRAN     BUFF     RIGHT     (L-ULD)
OR        M0261A	// OUT-BUFF MOVE->L (LEFT-P&P)
AND NOT   T2050	// OUT-TRAN     BUFF     LEFT     (R-ULD)
OUT       M0261A	// OUT-BUFF MOVE->L (LEFT-P&P)
// output comment: LEFT MOVE (LEFT P&P , RIGHT UNLOAD POSITION
; L20
LOAD      M02413	// L-R ALL AUTO
AND       T2055	// R_OUT BUFFER VC-NOTH
OR        M02410	// ONLY LEFT AUTO
LOAD      T2052	// L_OUT BUFFER VC ON
LOAD      M02413	// L-R ALL AUTO
AND       M12010	// L_P&P STEP#00
AND       M14515	// R_P&P STEP#05
OR LOAD
AND LOAD
LOAD      M02411	// ONLY RIGHT AUTO
AND       T2055	// R_OUT BUFFER VC-NOTH
OR LOAD
OR        M18864	// T)R_OUT BUFFER RIGHT
AND       M02614	// OUT-BUFF MOV SAFE
AND       T2050	// OUT-TRAN     BUFF     LEFT     (R-ULD)
OR        M0261B	// OUT-BUFF MOVE->R (RIGT-P&P)
AND NOT   T2051	// OUT-TRAN     BUFF     RIGHT     (L-ULD)
OUT       M0261B	// OUT-BUFF MOVE->R (RIGT-P&P)
// output comment: RIGHT MOVE (LEFT UNLOAD, RIGHT P&P POSITION
; L25
LOAD      M0261A	// OUT-BUFF MOVE->L (LEFT-P&P)
LOAD      M0241C	// IN-BUFF MOV->LEFT
AND       M0191A
OR LOAD
OUT       P0010E	// OUT_BUFF MOV L_P&P >

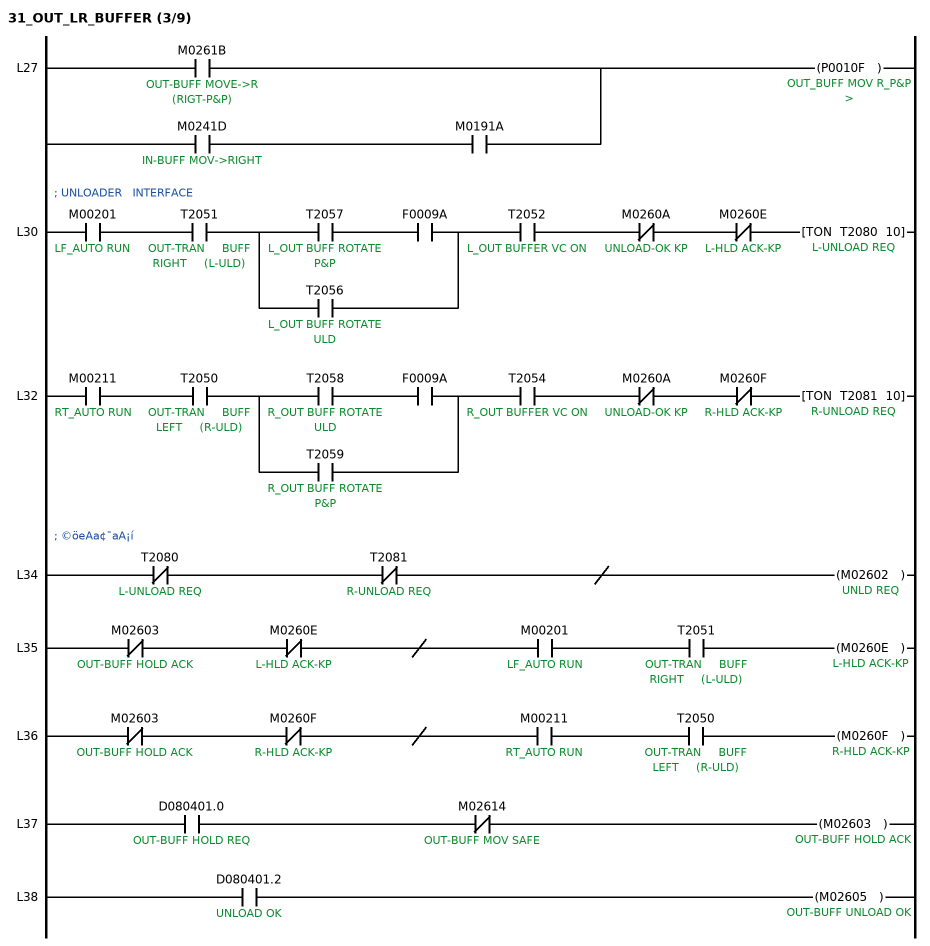
; L27
LOAD      M0261B	// OUT-BUFF MOVE->R (RIGT-P&P)
LOAD      M0241D	// IN-BUFF MOV->RIGHT
AND       M0191A
OR LOAD
OUT       P0010F	// OUT_BUFF MOV R_P&P >
//  UNLOADER   INTERFACE
; L30
LOAD      M00201	// LF_AUTO RUN
AND       T2051	// OUT-TRAN     BUFF     RIGHT     (L-ULD)
LOAD      T2057	// L_OUT BUFF ROTATE      P&P
AND       F0009A
OR        T2056	// L_OUT BUFF ROTATE     ULD
AND LOAD
AND       T2052	// L_OUT BUFFER VC ON
AND NOT   M0260A	// UNLOAD-OK KP
AND NOT   M0260E	// L-HLD ACK-KP
TON       T2080 10	// L-UNLOAD REQ
; L32
LOAD      M00211	// RT_AUTO RUN
AND       T2050	// OUT-TRAN     BUFF     LEFT     (R-ULD)
LOAD      T2058	// R_OUT BUFF ROTATE      ULD
AND       F0009A
OR        T2059	// R_OUT BUFF ROTATE      P&P
AND LOAD
AND       T2054	// R_OUT BUFFER VC ON
AND NOT   M0260A	// UNLOAD-OK KP
AND NOT   M0260F	// R-HLD ACK-KP
TON       T2081 10	// R-UNLOAD REQ
; L34
LOAD NOT  T2080	// L-UNLOAD REQ
AND NOT   T2081	// R-UNLOAD REQ
NOT
OUT       M02602	// UNLD REQ
// output comment: ©öeAa¢¯aA¡í
; L35
LOAD NOT  M02603	// OUT-BUFF HOLD ACK
AND NOT   M0260E	// L-HLD ACK-KP
NOT
AND       M00201	// LF_AUTO RUN
AND       T2051	// OUT-TRAN     BUFF     RIGHT     (L-ULD)
OUT       M0260E	// L-HLD ACK-KP
; L36
LOAD NOT  M02603	// OUT-BUFF HOLD ACK
AND NOT   M0260F	// R-HLD ACK-KP
NOT
AND       M00211	// RT_AUTO RUN
AND       T2050	// OUT-TRAN     BUFF     LEFT     (R-ULD)
OUT       M0260F	// R-HLD ACK-KP
; L37
LOAD      D080401.0	// OUT-BUFF HOLD REQ
AND NOT   M02614	// OUT-BUFF MOV SAFE
OUT       M02603	// OUT-BUFF HOLD ACK
; L38
LOAD      D080401.2	// UNLOAD OK
OUT       M02605	// OUT-BUFF UNLOAD OK

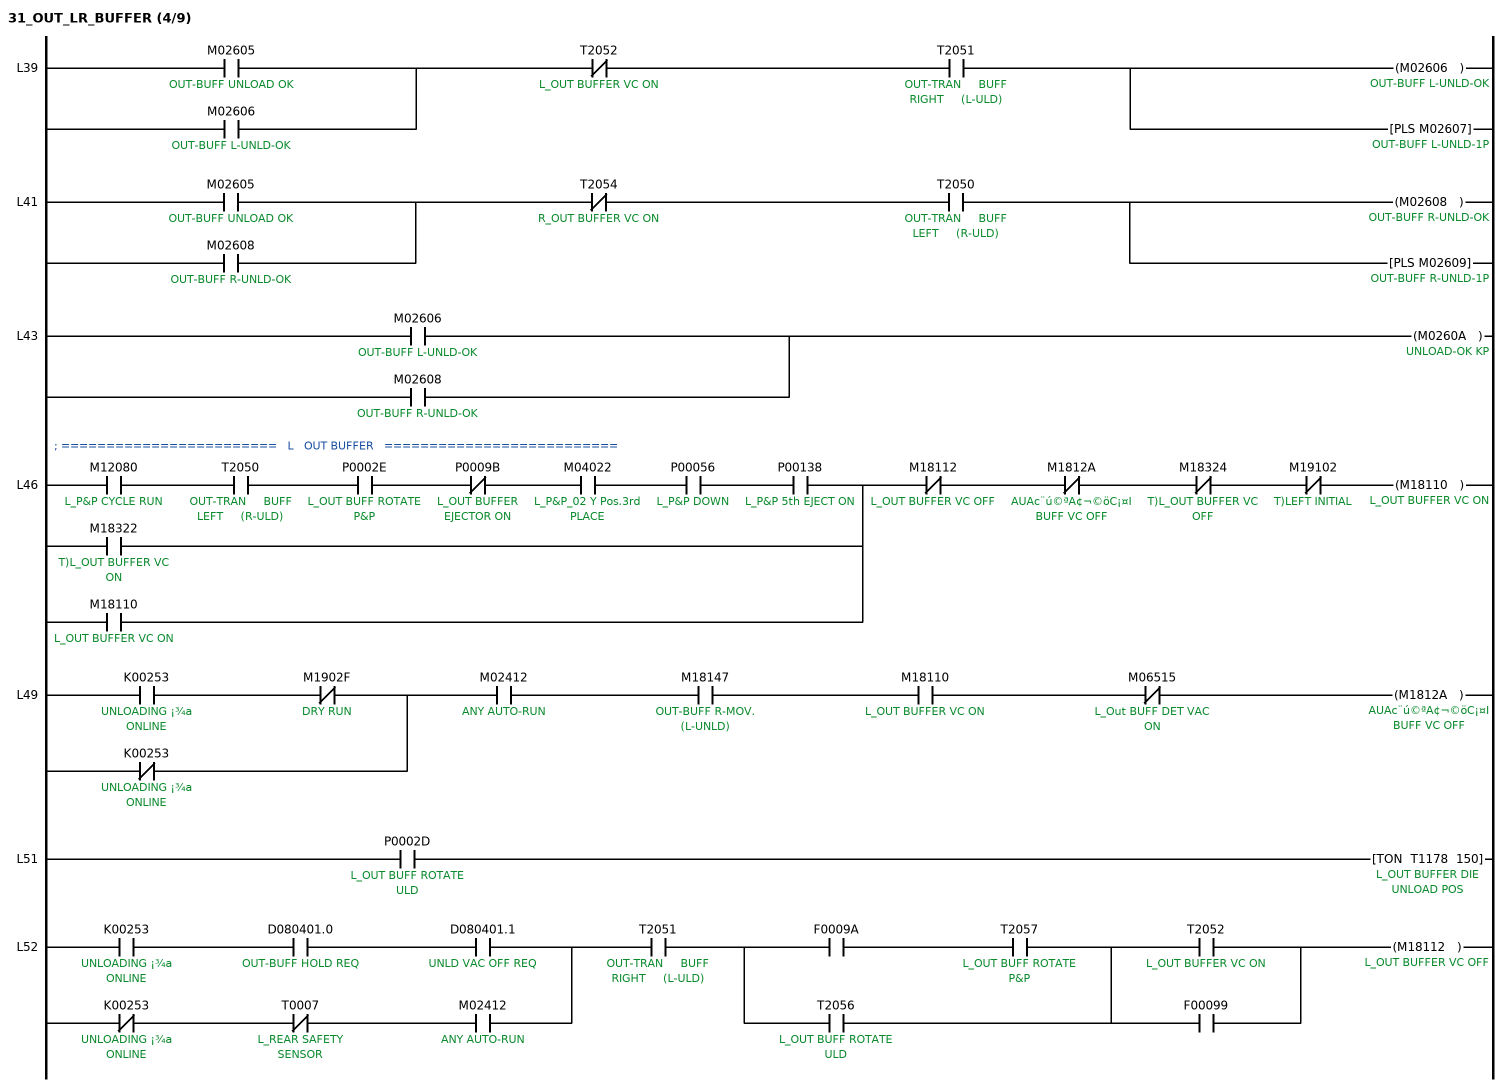
; L39
LOAD      M02605	// OUT-BUFF UNLOAD OK
OR        M02606	// OUT-BUFF L-UNLD-OK
AND NOT   T2052	// L_OUT BUFFER VC ON
AND       T2051	// OUT-TRAN     BUFF     RIGHT     (L-ULD)
OUT       M02606	// OUT-BUFF L-UNLD-OK
OUTP      M02607	// OUT-BUFF L-UNLD-1P
; L41
LOAD      M02605	// OUT-BUFF UNLOAD OK
OR        M02608	// OUT-BUFF R-UNLD-OK
AND NOT   T2054	// R_OUT BUFFER VC ON
AND       T2050	// OUT-TRAN     BUFF     LEFT     (R-ULD)
OUT       M02608	// OUT-BUFF R-UNLD-OK
OUTP      M02609	// OUT-BUFF R-UNLD-1P
; L43
LOAD      M02606	// OUT-BUFF L-UNLD-OK
OR        M02608	// OUT-BUFF R-UNLD-OK
OUT       M0260A	// UNLOAD-OK KP
// ========================   L   OUT BUFFER   ==========================
; L46
LOAD      M12080	// L_P&P CYCLE RUN
AND       T2050	// OUT-TRAN     BUFF     LEFT     (R-ULD)
AND       P0002E	// L_OUT BUFF ROTATE      P&P
AND NOT   P0009B	// L_OUT BUFFER EJECTOR ON
AND       M04022	// L_P&P_02 Y Pos.3rd PLACE
AND       P00056	// L_P&P DOWN
AND       P00138	// L_P&P 5th EJECT ON
OR        M18322	// T)L_OUT BUFFER VC ON
OR        M18110	// L_OUT BUFFER VC ON
AND NOT   M18112	// L_OUT BUFFER VC OFF
AND NOT   M1812A	// AUAc¨ú©ªA¢¬©öC¡¤I BUFF VC OFF
AND NOT   M18324	// T)L_OUT BUFFER VC OFF
AND NOT   M19102	// T)LEFT INITIAL
OUT       M18110	// L_OUT BUFFER VC ON
; L49
LOAD      K00253	// UNLOADING ¡¾a ONLINE
AND NOT   M1902F	// DRY RUN
OR NOT    K00253	// UNLOADING ¡¾a ONLINE
AND       M02412	// ANY AUTO-RUN
AND       M18147	// OUT-BUFF R-MOV.  (L-UNLD)
AND       M18110	// L_OUT BUFFER VC ON
AND NOT   M06515	// L_Out BUFF DET VAC ON
OUT       M1812A	// AUAc¨ú©ªA¢¬©öC¡¤I BUFF VC OFF
; L51
LOAD      P0002D	// L_OUT BUFF ROTATE     ULD
TON       T1178 150	// L_OUT BUFFER DIE UNLOAD POS
; L52
LOAD      K00253	// UNLOADING ¡¾a ONLINE
AND       D080401.0	// OUT-BUFF HOLD REQ
AND       D080401.1	// UNLD VAC OFF REQ
LOAD NOT  K00253	// UNLOADING ¡¾a ONLINE
AND NOT   T0007	// L_REAR SAFETY SENSOR
AND       M02412	// ANY AUTO-RUN
OR LOAD
AND       T2051	// OUT-TRAN     BUFF     RIGHT     (L-ULD)
LOAD      F0009A
AND       T2057	// L_OUT BUFF ROTATE      P&P
OR        T2056	// L_OUT BUFF ROTATE     ULD
AND LOAD
LOAD      T2052	// L_OUT BUFFER VC ON
OR        F00099
AND LOAD
OUT       M18112	// L_OUT BUFFER VC OFF

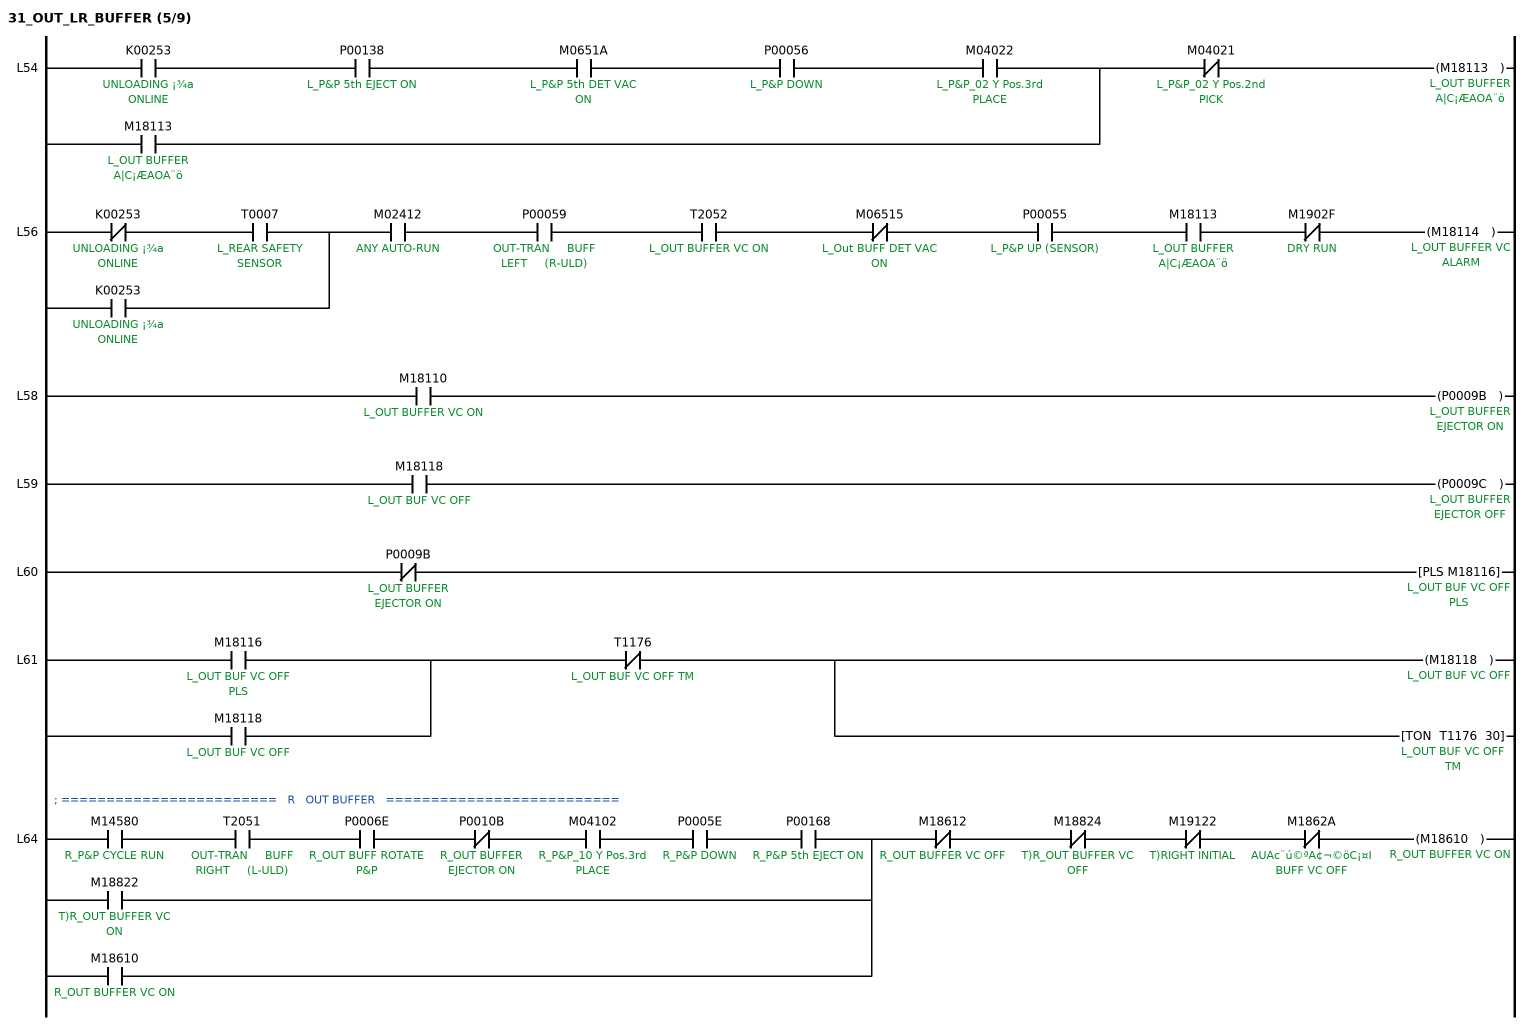
; L54
LOAD      K00253	// UNLOADING ¡¾a ONLINE
AND       P00138	// L_P&P 5th EJECT ON
AND       M0651A	// L_P&P 5th DET VAC ON
AND       P00056	// L_P&P DOWN
AND       M04022	// L_P&P_02 Y Pos.3rd PLACE
OR        M18113	// L_OUT BUFFER A|C¡ÆAOA¨ö
AND NOT   M04021	// L_P&P_02 Y Pos.2nd PICK
OUT       M18113	// L_OUT BUFFER A|C¡ÆAOA¨ö
; L56
LOAD NOT  K00253	// UNLOADING ¡¾a ONLINE
AND       T0007	// L_REAR SAFETY SENSOR
OR        K00253	// UNLOADING ¡¾a ONLINE
AND       M02412	// ANY AUTO-RUN
AND       P00059	// OUT-TRAN     BUFF     LEFT     (R-ULD)
AND       T2052	// L_OUT BUFFER VC ON
AND NOT   M06515	// L_Out BUFF DET VAC ON
AND       P00055	// L_P&P UP (SENSOR)
AND       M18113	// L_OUT BUFFER A|C¡ÆAOA¨ö
AND NOT   M1902F	// DRY RUN
OUT       M18114	// L_OUT BUFFER VC ALARM
; L58
LOAD      M18110	// L_OUT BUFFER VC ON
OUT       P0009B	// L_OUT BUFFER EJECTOR ON
; L59
LOAD      M18118	// L_OUT BUF VC OFF
OUT       P0009C	// L_OUT BUFFER EJECTOR OFF
; L60
LOAD NOT  P0009B	// L_OUT BUFFER EJECTOR ON
OUTP      M18116	// L_OUT BUF VC OFF PLS
; L61
LOAD      M18116	// L_OUT BUF VC OFF PLS
OR        M18118	// L_OUT BUF VC OFF
AND NOT   T1176	// L_OUT BUF VC OFF TM
OUT       M18118	// L_OUT BUF VC OFF
TON       T1176 30	// L_OUT BUF VC OFF TM
// ========================   R   OUT BUFFER   ==========================
; L64
LOAD      M14580	// R_P&P CYCLE RUN
AND       T2051	// OUT-TRAN     BUFF     RIGHT     (L-ULD)
AND       P0006E	// R_OUT BUFF ROTATE      P&P
AND NOT   P0010B	// R_OUT BUFFER EJECTOR ON
AND       M04102	// R_P&P_10 Y Pos.3rd PLACE
AND       P0005E	// R_P&P DOWN
AND       P00168	// R_P&P 5th EJECT ON
OR        M18822	// T)R_OUT BUFFER VC ON
OR        M18610	// R_OUT BUFFER VC ON
AND NOT   M18612	// R_OUT BUFFER VC OFF
AND NOT   M18824	// T)R_OUT BUFFER VC OFF
AND NOT   M19122	// T)RIGHT INITIAL
AND NOT   M1862A	// AUAc¨ú©ªA¢¬©öC¡¤I BUFF VC OFF
OUT       M18610	// R_OUT BUFFER VC ON

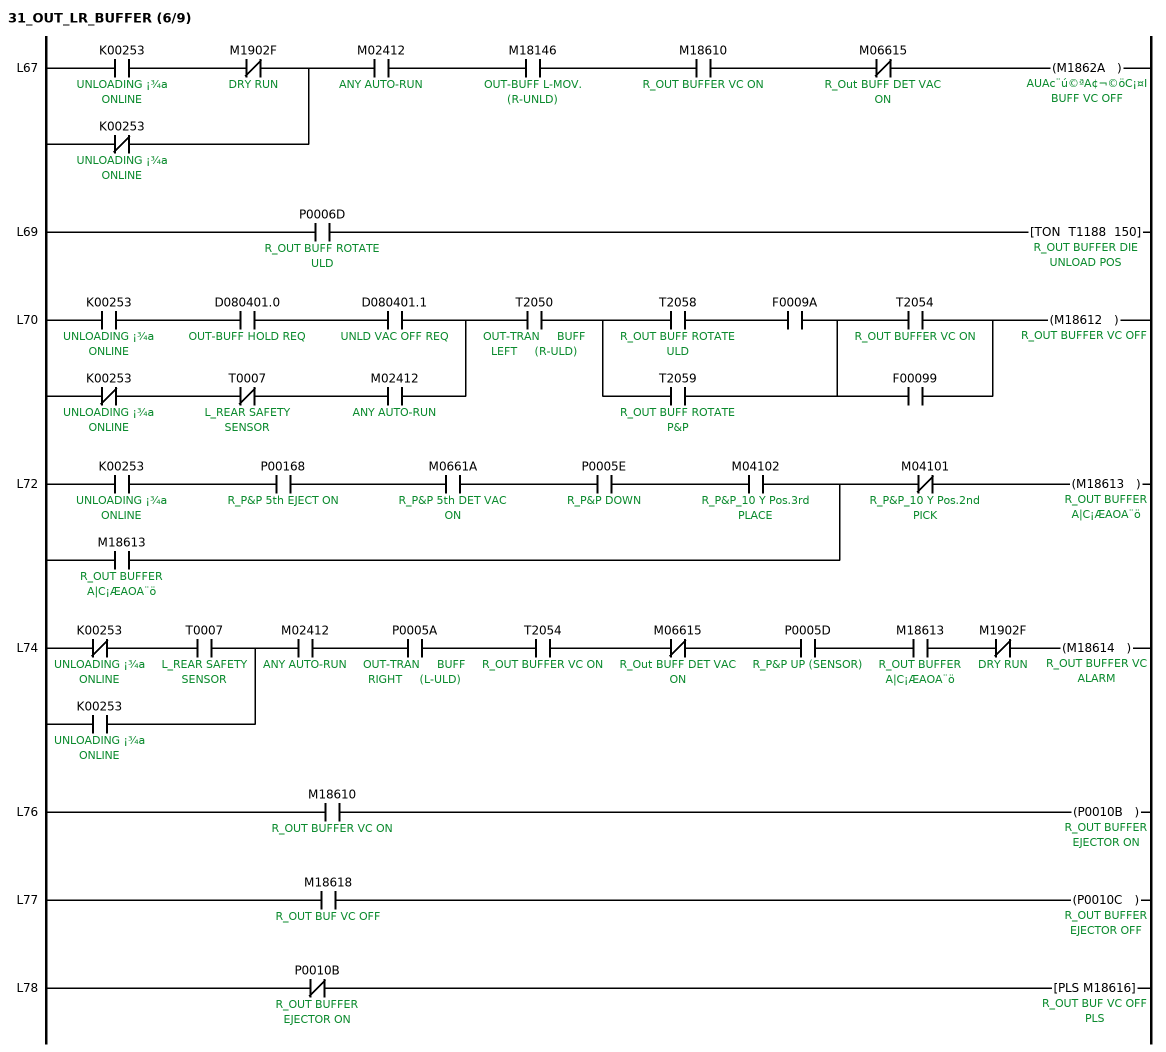
; L67
LOAD      K00253	// UNLOADING ¡¾a ONLINE
AND NOT   M1902F	// DRY RUN
OR NOT    K00253	// UNLOADING ¡¾a ONLINE
AND       M02412	// ANY AUTO-RUN
AND       M18146	// OUT-BUFF L-MOV.  (R-UNLD)
AND       M18610	// R_OUT BUFFER VC ON
AND NOT   M06615	// R_Out BUFF DET VAC ON
OUT       M1862A	// AUAc¨ú©ªA¢¬©öC¡¤I BUFF VC OFF
; L69
LOAD      P0006D	// R_OUT BUFF ROTATE      ULD
TON       T1188 150	// R_OUT BUFFER DIE UNLOAD POS
; L70
LOAD      K00253	// UNLOADING ¡¾a ONLINE
AND       D080401.0	// OUT-BUFF HOLD REQ
AND       D080401.1	// UNLD VAC OFF REQ
LOAD NOT  K00253	// UNLOADING ¡¾a ONLINE
AND NOT   T0007	// L_REAR SAFETY SENSOR
AND       M02412	// ANY AUTO-RUN
OR LOAD
AND       T2050	// OUT-TRAN     BUFF     LEFT     (R-ULD)
LOAD      T2058	// R_OUT BUFF ROTATE      ULD
AND       F0009A
OR        T2059	// R_OUT BUFF ROTATE      P&P
AND LOAD
LOAD      T2054	// R_OUT BUFFER VC ON
OR        F00099
AND LOAD
OUT       M18612	// R_OUT BUFFER VC OFF
; L72
LOAD      K00253	// UNLOADING ¡¾a ONLINE
AND       P00168	// R_P&P 5th EJECT ON
AND       M0661A	// R_P&P 5th DET VAC ON
AND       P0005E	// R_P&P DOWN
AND       M04102	// R_P&P_10 Y Pos.3rd PLACE
OR        M18613	// R_OUT BUFFER A|C¡ÆAOA¨ö
AND NOT   M04101	// R_P&P_10 Y Pos.2nd PICK
OUT       M18613	// R_OUT BUFFER A|C¡ÆAOA¨ö
; L74
LOAD NOT  K00253	// UNLOADING ¡¾a ONLINE
AND       T0007	// L_REAR SAFETY SENSOR
OR        K00253	// UNLOADING ¡¾a ONLINE
AND       M02412	// ANY AUTO-RUN
AND       P0005A	// OUT-TRAN     BUFF     RIGHT     (L-ULD)
AND       T2054	// R_OUT BUFFER VC ON
AND NOT   M06615	// R_Out BUFF DET VAC ON
AND       P0005D	// R_P&P UP (SENSOR)
AND       M18613	// R_OUT BUFFER A|C¡ÆAOA¨ö
AND NOT   M1902F	// DRY RUN
OUT       M18614	// R_OUT BUFFER VC ALARM
; L76
LOAD      M18610	// R_OUT BUFFER VC ON
OUT       P0010B	// R_OUT BUFFER EJECTOR ON
; L77
LOAD      M18618	// R_OUT BUF VC OFF
OUT       P0010C	// R_OUT BUFFER EJECTOR OFF
; L78
LOAD NOT  P0010B	// R_OUT BUFFER EJECTOR ON
OUTP      M18616	// R_OUT BUF VC OFF PLS

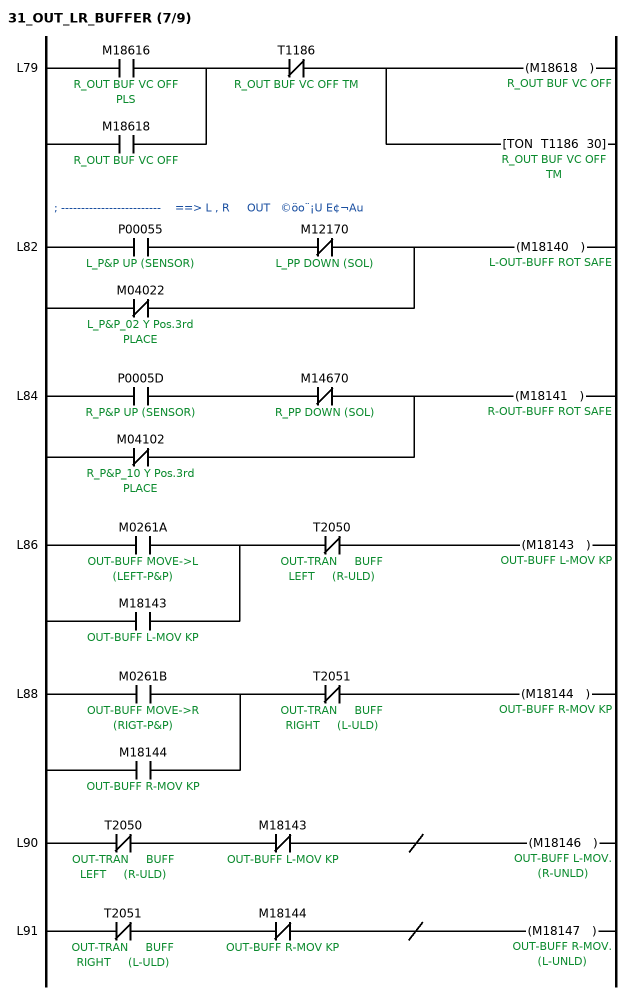
; L79
LOAD      M18616	// R_OUT BUF VC OFF PLS
OR        M18618	// R_OUT BUF VC OFF
AND NOT   T1186	// R_OUT BUF VC OFF TM
OUT       M18618	// R_OUT BUF VC OFF
TON       T1186 30	// R_OUT BUF VC OFF TM
// -------------------------    ==> L , R     OUT   ©öo¨¡U E¢¬Au
; L82
LOAD      P00055	// L_P&P UP (SENSOR)
AND NOT   M12170	// L_PP DOWN (SOL)
OR NOT    M04022	// L_P&P_02 Y Pos.3rd PLACE
OUT       M18140	// L-OUT-BUFF ROT SAFE
; L84
LOAD      P0005D	// R_P&P UP (SENSOR)
AND NOT   M14670	// R_PP DOWN (SOL)
OR NOT    M04102	// R_P&P_10 Y Pos.3rd PLACE
OUT       M18141	// R-OUT-BUFF ROT SAFE
; L86
LOAD      M0261A	// OUT-BUFF MOVE->L (LEFT-P&P)
OR        M18143	// OUT-BUFF L-MOV KP
AND NOT   T2050	// OUT-TRAN     BUFF     LEFT     (R-ULD)
OUT       M18143	// OUT-BUFF L-MOV KP
; L88
LOAD      M0261B	// OUT-BUFF MOVE->R (RIGT-P&P)
OR        M18144	// OUT-BUFF R-MOV KP
AND NOT   T2051	// OUT-TRAN     BUFF     RIGHT     (L-ULD)
OUT       M18144	// OUT-BUFF R-MOV KP
; L90
LOAD NOT  T2050	// OUT-TRAN     BUFF     LEFT     (R-ULD)
AND NOT   M18143	// OUT-BUFF L-MOV KP
NOT
OUT       M18146	// OUT-BUFF L-MOV.  (R-UNLD)
; L91
LOAD NOT  T2051	// OUT-TRAN     BUFF     RIGHT     (L-ULD)
AND NOT   M18144	// OUT-BUFF R-MOV KP
NOT
OUT       M18147	// OUT-BUFF R-MOV.  (L-UNLD)

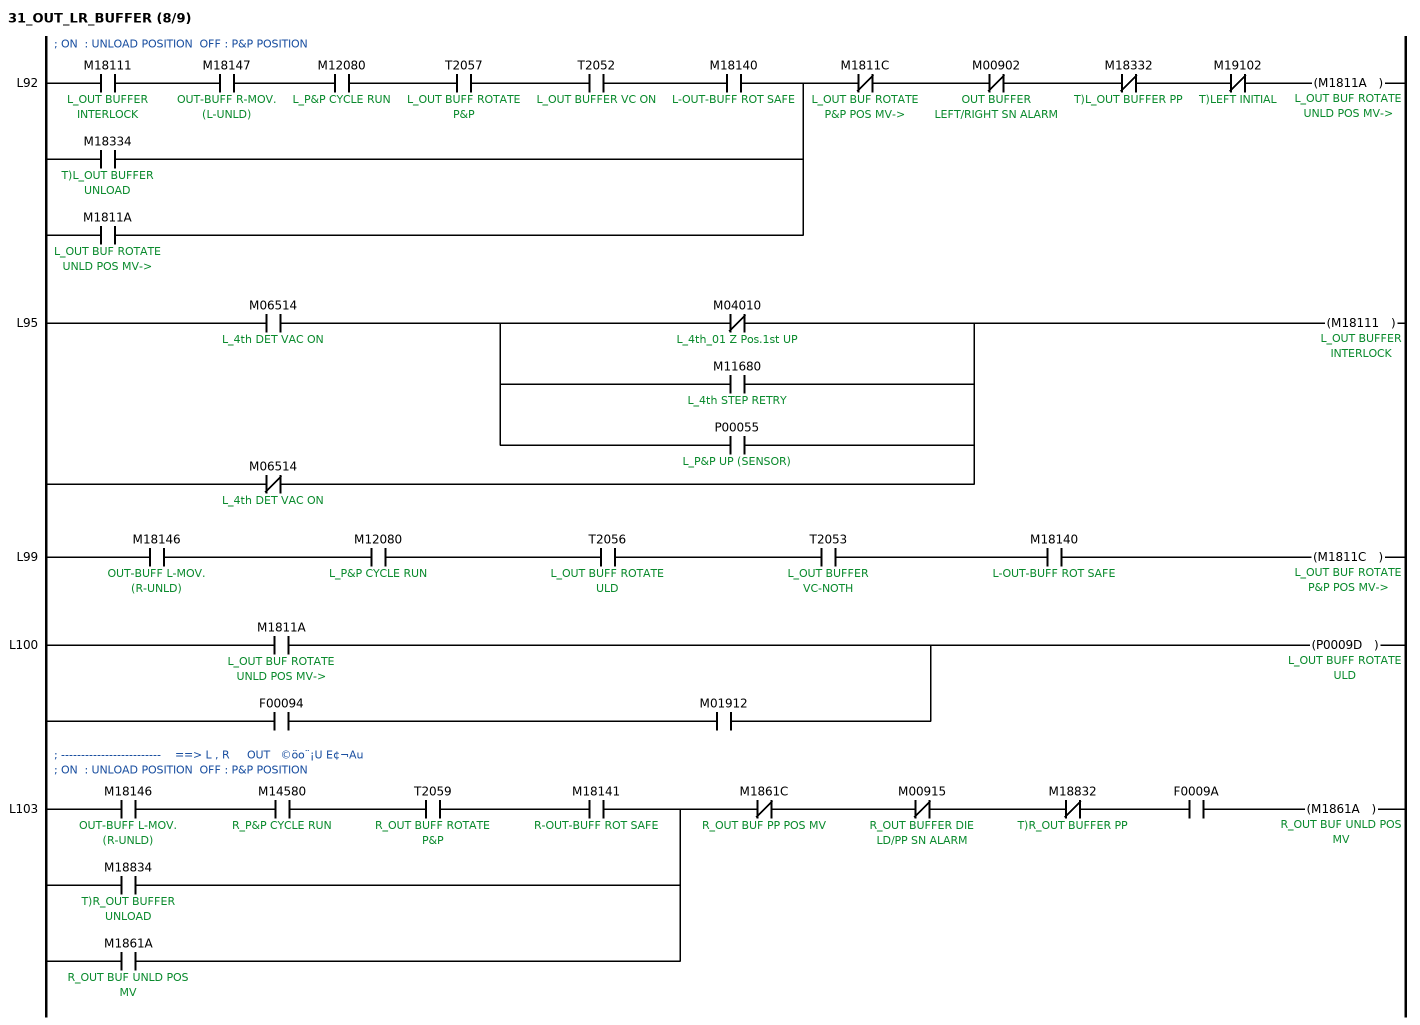
; L92
LOAD      M18111	// L_OUT BUFFER INTERLOCK
AND       M18147	// OUT-BUFF R-MOV.  (L-UNLD)
AND       M12080	// L_P&P CYCLE RUN
AND       T2057	// L_OUT BUFF ROTATE      P&P
AND       T2052	// L_OUT BUFFER VC ON
AND       M18140	// L-OUT-BUFF ROT SAFE
OR        M18334	// T)L_OUT BUFFER UNLOAD
OR        M1811A	// L_OUT BUF ROTATE UNLD POS MV->
AND NOT   M1811C	// L_OUT BUF ROTATE P&P POS MV->
AND NOT   M00902	// OUT BUFFER LEFT/RIGHT SN ALARM
AND NOT   M18332	// T)L_OUT BUFFER PP
AND NOT   M19102	// T)LEFT INITIAL
OUT       M1811A	// L_OUT BUF ROTATE UNLD POS MV->
// output comment: ON  : UNLOAD POSITION  OFF : P&P POSITION
; L95
LOAD      M06514	// L_4th DET VAC ON
LOAD NOT  M04010	// L_4th_01 Z Pos.1st UP
OR        M11680	// L_4th STEP RETRY
OR        P00055	// L_P&P UP (SENSOR)
AND LOAD
OR NOT    M06514	// L_4th DET VAC ON
OUT       M18111	// L_OUT BUFFER INTERLOCK
; L99
LOAD      M18146	// OUT-BUFF L-MOV.  (R-UNLD)
AND       M12080	// L_P&P CYCLE RUN
AND       T2056	// L_OUT BUFF ROTATE     ULD
AND       T2053	// L_OUT BUFFER VC-NOTH
AND       M18140	// L-OUT-BUFF ROT SAFE
OUT       M1811C	// L_OUT BUF ROTATE P&P POS MV->
; L100
LOAD      M1811A	// L_OUT BUF ROTATE UNLD POS MV->
LOAD      F00094
AND       M01912
OR LOAD
OUT       P0009D	// L_OUT BUFF ROTATE ULD
// -------------------------    ==> L , R     OUT   ©öo¨¡U E¢¬Au
; L103
LOAD      M18146	// OUT-BUFF L-MOV.  (R-UNLD)
AND       M14580	// R_P&P CYCLE RUN
AND       T2059	// R_OUT BUFF ROTATE      P&P
AND       M18141	// R-OUT-BUFF ROT SAFE
OR        M18834	// T)R_OUT BUFFER UNLOAD
OR        M1861A	// R_OUT BUF UNLD POS MV
AND NOT   M1861C	// R_OUT BUF PP POS MV
AND NOT   M00915	// R_OUT BUFFER DIE LD/PP SN ALARM
AND NOT   M18832	// T)R_OUT BUFFER PP
AND       F0009A
OUT       M1861A	// R_OUT BUF UNLD POS MV
// output comment: ON  : UNLOAD POSITION  OFF : P&P POSITION

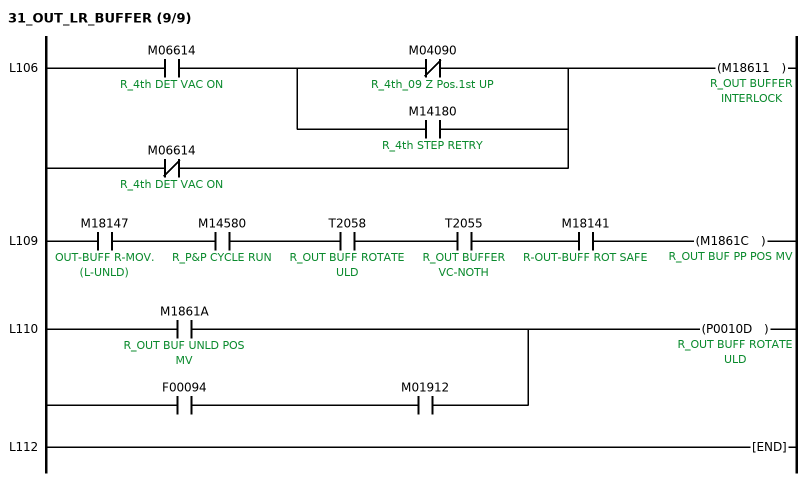
; L106
LOAD      M06614	// R_4th DET VAC ON
LOAD NOT  M04090	// R_4th_09 Z Pos.1st UP
OR        M14180	// R_4th STEP RETRY
AND LOAD
OR NOT    M06614	// R_4th DET VAC ON
OUT       M18611	// R_OUT BUFFER INTERLOCK
; L109
LOAD      M18147	// OUT-BUFF R-MOV.  (L-UNLD)
AND       M14580	// R_P&P CYCLE RUN
AND       T2058	// R_OUT BUFF ROTATE      ULD
AND       T2055	// R_OUT BUFFER VC-NOTH
AND       M18141	// R-OUT-BUFF ROT SAFE
OUT       M1861C	// R_OUT BUF PP POS MV
; L110
LOAD      M1861A	// R_OUT BUF UNLD POS MV
LOAD      F00094
AND       M01912
OR LOAD
OUT       P0010D	// R_OUT BUFF ROTATE ULD
; L112
END

PROGRAM 40_2D_CODE (task: ¨ö¨¬A¥ì CA¡¤I¡¾¡¿¡¤¡Í)

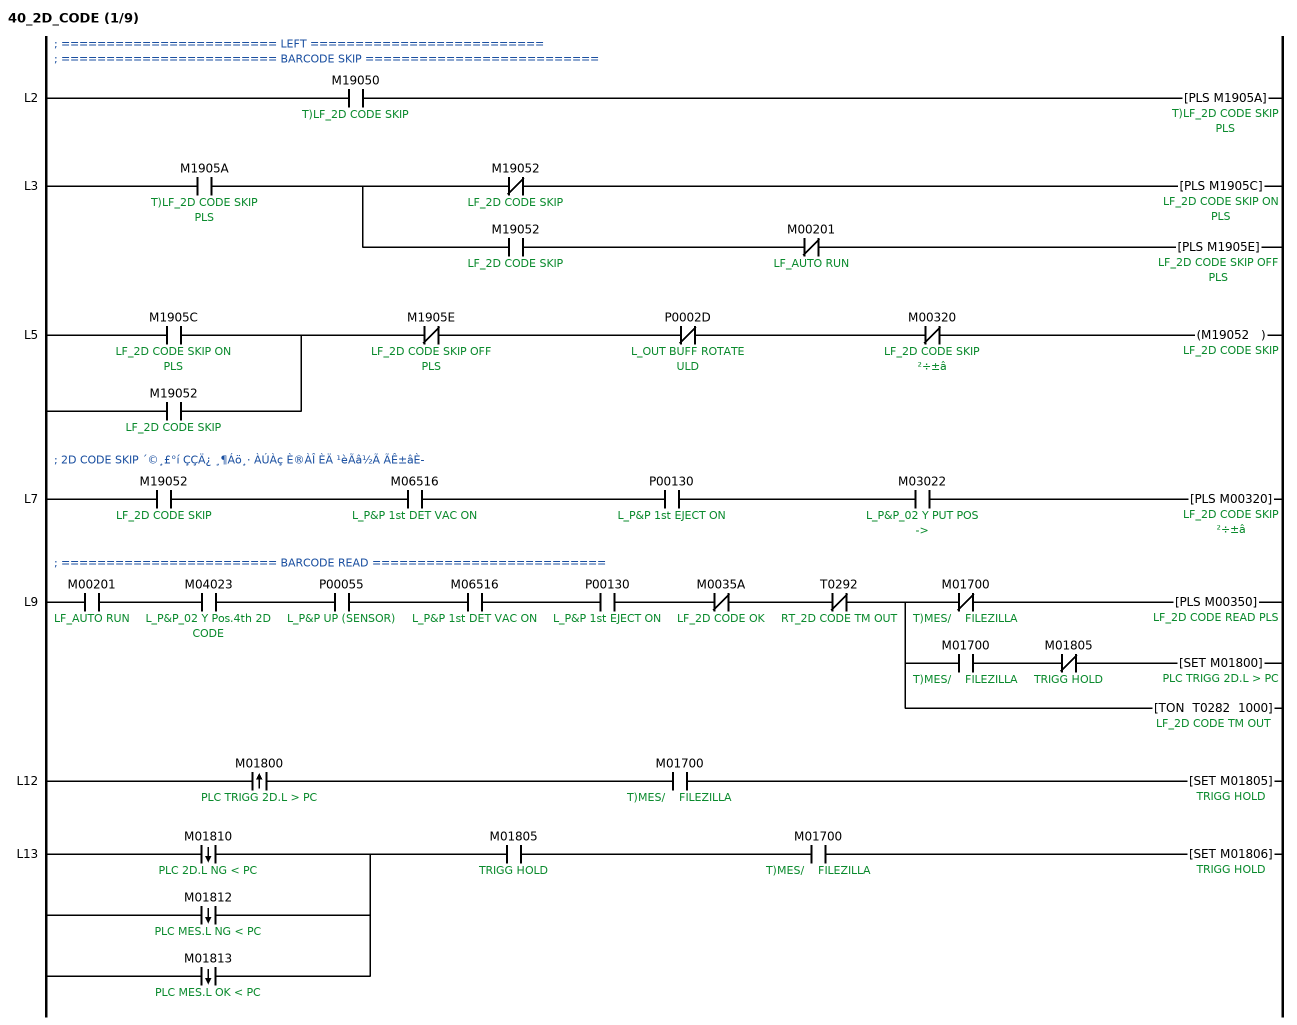
// ======================== LEFT ==========================
// ======================== BARCODE SKIP ==========================
; L2
LOAD      M19050	// T)LF_2D CODE SKIP
OUTP      M1905A	// T)LF_2D CODE SKIP PLS
; L3
LOAD      M1905A	// T)LF_2D CODE SKIP PLS
MPUSH
AND NOT   M19052	// LF_2D CODE SKIP
OUTP      M1905C	// LF_2D CODE SKIP ON PLS
MPOP
AND       M19052	// LF_2D CODE SKIP
AND NOT   M00201	// LF_AUTO RUN
OUTP      M1905E	// LF_2D CODE SKIP OFF PLS
; L5
LOAD      M1905C	// LF_2D CODE SKIP ON PLS
OR        M19052	// LF_2D CODE SKIP
AND NOT   M1905E	// LF_2D CODE SKIP OFF PLS
AND NOT   P0002D	// L_OUT BUFF ROTATE     ULD
AND NOT   M00320	// LF_2D CODE SKIP ²÷±â
OUT       M19052	// LF_2D CODE SKIP
; L7
LOAD      M19052	// LF_2D CODE SKIP
AND       M06516	// L_P&P 1st DET VAC ON
AND       P00130	// L_P&P 1st EJECT ON
AND       M03022	// L_P&P_02 Y PUT POS ->
OUTP      M00320	// LF_2D CODE SKIP ²÷±â
// output comment: 2D CODE SKIP ´©¸£°í ÇÇÄ¿ ¸¶Áö¸· ÀÚÀç È®ÀÎ ÈÄ ¹èÃâ½Ã ÃÊ±âÈ­
// ======================== BARCODE READ ==========================
; L9
LOAD      M00201	// LF_AUTO RUN
AND       M04023	// L_P&P_02 Y Pos.4th 2D CODE
AND       P00055	// L_P&P UP (SENSOR)
AND       M06516	// L_P&P 1st DET VAC ON
AND       P00130	// L_P&P 1st EJECT ON
AND NOT   M0035A	// LF_2D CODE OK
AND NOT   T0292	// RT_2D CODE TM OUT
MPUSH
AND NOT   M01700	// T)MES/    FILEZILLA
OUTP      M00350	// LF_2D CODE READ PLS
MLOAD
AND       M01700	// T)MES/    FILEZILLA
AND NOT   M01805	// TRIGG HOLD
SET       M01800	// PLC TRIGG 2D.L > PC
MPOP
TON       T0282 1000	// LF_2D CODE TM OUT
; L12
LOADP     M01800	// PLC TRIGG 2D.L > PC
AND       M01700	// T)MES/    FILEZILLA
SET       M01805	// TRIGG HOLD
; L13
LOADN     M01810	// PLC 2D.L NG < PC
ORN       M01812	// PLC MES.L NG < PC
ORN       M01813	// PLC MES.L OK < PC
AND       M01805	// TRIGG HOLD
AND       M01700	// T)MES/    FILEZILLA
SET       M01806	// TRIGG HOLD

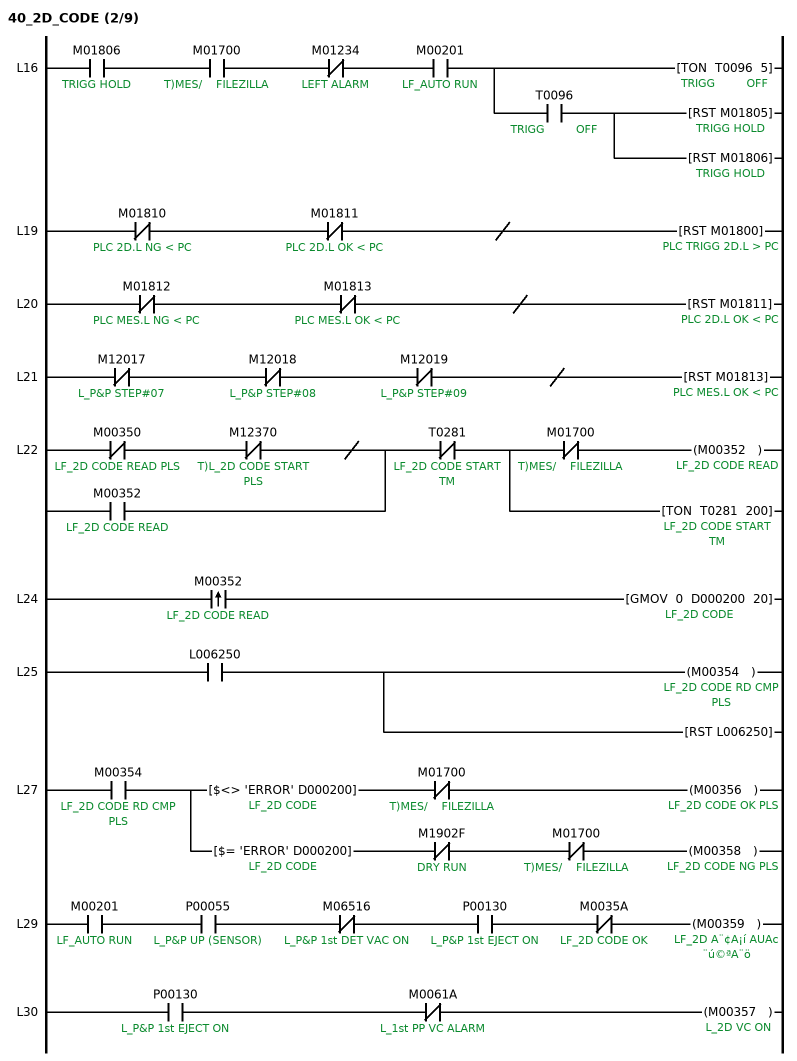
; L16
LOAD      M01806	// TRIGG HOLD
AND       M01700	// T)MES/    FILEZILLA
AND NOT   M01234	// LEFT ALARM
AND       M00201	// LF_AUTO RUN
TON       T0096 5	// TRIGG         OFF
AND       T0096	// TRIGG         OFF
RST       M01805	// TRIGG HOLD
RST       M01806	// TRIGG HOLD
; L19
LOAD NOT  M01810	// PLC 2D.L NG < PC
AND NOT   M01811	// PLC 2D.L OK < PC
NOT
RST       M01800	// PLC TRIGG 2D.L > PC
; L20
LOAD NOT  M01812	// PLC MES.L NG < PC
AND NOT   M01813	// PLC MES.L OK < PC
NOT
RST       M01811	// PLC 2D.L OK < PC
; L21
LOAD NOT  M12017	// L_P&P STEP#07
AND NOT   M12018	// L_P&P STEP#08
AND NOT   M12019	// L_P&P STEP#09
NOT
RST       M01813	// PLC MES.L OK < PC
; L22
LOAD NOT  M00350	// LF_2D CODE READ PLS
AND NOT   M12370	// T)L_2D CODE START PLS
NOT
OR        M00352	// LF_2D CODE READ
AND NOT   T0281	// LF_2D CODE START TM
MPUSH
AND NOT   M01700	// T)MES/    FILEZILLA
OUT       M00352	// LF_2D CODE READ
MPOP
TON       T0281 200	// LF_2D CODE START TM
; L24
LOADP     M00352	// LF_2D CODE READ
GMOV      0 D000200 20	// LF_2D CODE
; L25
LOAD      L006250
OUT       M00354	// LF_2D CODE RD CMP PLS
RST       L006250
; L27
LOAD      M00354	// LF_2D CODE RD CMP PLS
MPUSH
AND$<>    'ERROR' D000200	// LF_2D CODE
AND NOT   M01700	// T)MES/    FILEZILLA
OUT       M00356	// LF_2D CODE OK PLS
MPOP
AND$=     'ERROR' D000200	// LF_2D CODE
AND NOT   M1902F	// DRY RUN
AND NOT   M01700	// T)MES/    FILEZILLA
OUT       M00358	// LF_2D CODE NG PLS
; L29
LOAD      M00201	// LF_AUTO RUN
AND       P00055	// L_P&P UP (SENSOR)
AND NOT   M06516	// L_P&P 1st DET VAC ON
AND       P00130	// L_P&P 1st EJECT ON
AND NOT   M0035A	// LF_2D CODE OK
OUT       M00359	// LF_2D A¨¢A¡í AUAc ¨ú©ªA¨ö
; L30
LOAD      P00130	// L_P&P 1st EJECT ON
AND NOT   M0061A	// L_1st PP VC ALARM
OUT       M00357	// L_2D VC ON

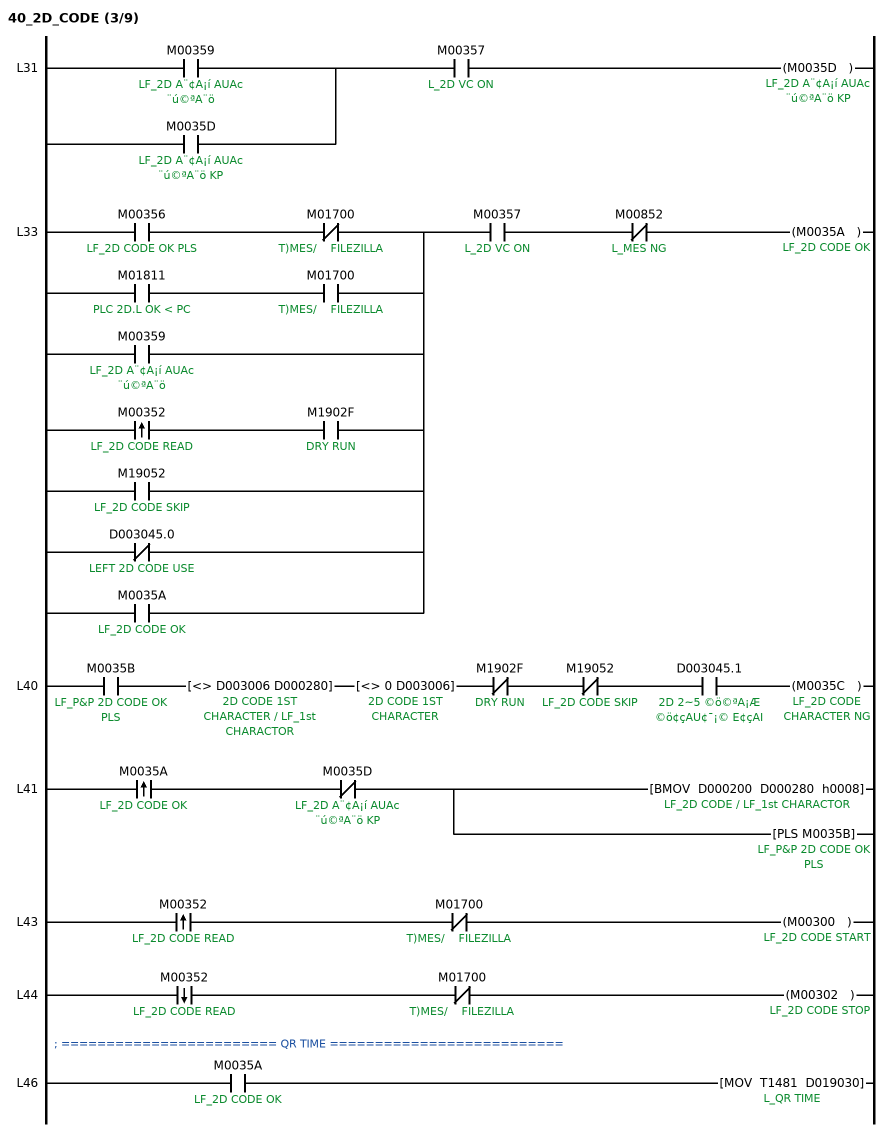
; L31
LOAD      M00359	// LF_2D A¨¢A¡í AUAc ¨ú©ªA¨ö
OR        M0035D	// LF_2D A¨¢A¡í AUAc ¨ú©ªA¨ö KP
AND       M00357	// L_2D VC ON
OUT       M0035D	// LF_2D A¨¢A¡í AUAc ¨ú©ªA¨ö KP
; L33
LOAD      M00356	// LF_2D CODE OK PLS
AND NOT   M01700	// T)MES/    FILEZILLA
LOAD      M01811	// PLC 2D.L OK < PC
AND       M01700	// T)MES/    FILEZILLA
OR LOAD
OR        M00359	// LF_2D A¨¢A¡í AUAc ¨ú©ªA¨ö
LOADP     M00352	// LF_2D CODE READ
AND       M1902F	// DRY RUN
OR LOAD
OR        M19052	// LF_2D CODE SKIP
OR NOT    D003045.0	// LEFT 2D CODE USE
OR        M0035A	// LF_2D CODE OK
AND       M00357	// L_2D VC ON
AND NOT   M00852	// L_MES NG
OUT       M0035A	// LF_2D CODE OK
; L40
LOAD      M0035B	// LF_P&P 2D CODE OK PLS
AND<>     D003006 D000280	// 2D CODE 1ST CHARACTER / LF_1st CHARACTOR
AND<>     0 D003006	// 2D CODE 1ST CHARACTER
AND NOT   M1902F	// DRY RUN
AND NOT   M19052	// LF_2D CODE SKIP
AND       D003045.1	// 2D 2~5 ©ö©ªA¡Æ ©ö¢çAU¢¯¡© E¢çAI
OUT       M0035C	// LF_2D CODE CHARACTER NG
; L41
LOADP     M0035A	// LF_2D CODE OK
AND NOT   M0035D	// LF_2D A¨¢A¡í AUAc ¨ú©ªA¨ö KP
BMOV      D000200 D000280 h0008	// LF_2D CODE / LF_1st CHARACTOR
OUTP      M0035B	// LF_P&P 2D CODE OK PLS
; L43
LOADP     M00352	// LF_2D CODE READ
AND NOT   M01700	// T)MES/    FILEZILLA
OUT       M00300	// LF_2D CODE START
; L44
LOADN     M00352	// LF_2D CODE READ
AND NOT   M01700	// T)MES/    FILEZILLA
OUT       M00302	// LF_2D CODE STOP
// ======================== QR TIME ==========================
; L46
LOAD      M0035A	// LF_2D CODE OK
MOV       T1481 D019030	// L_QR TIME

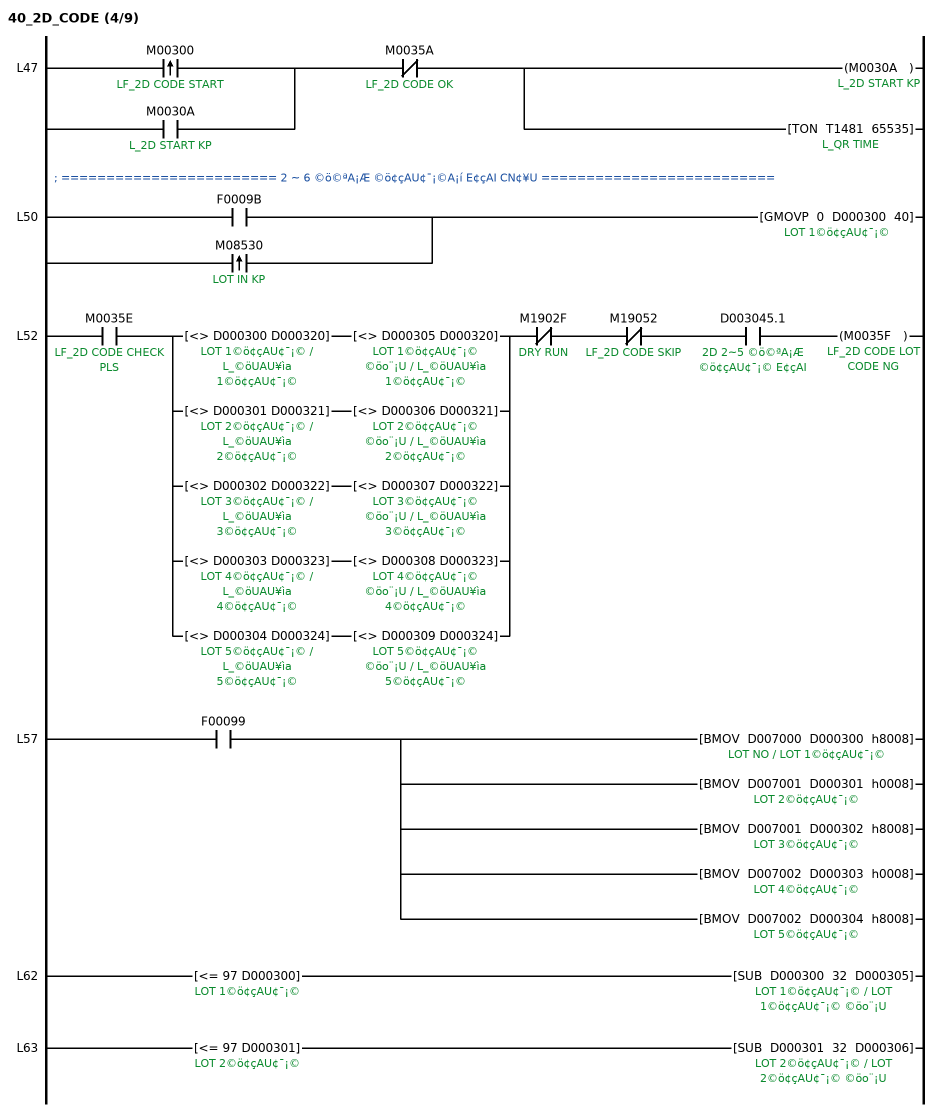
; L47
LOADP     M00300	// LF_2D CODE START
OR        M0030A	// L_2D START KP
AND NOT   M0035A	// LF_2D CODE OK
OUT       M0030A	// L_2D START KP
TON       T1481 65535	// L_QR TIME
// ======================== 2 ~ 6 ©ö©ªA¡Æ ©ö¢çAU¢¯¡©A¡í E¢çAI CN¢¥U ==========================
; L50
LOAD      F0009B
ORP       M08530	// LOT IN KP
GMOVP     0 D000300 40	// LOT 1©ö¢çAU¢¯¡©
; L52
LOAD      M0035E	// LF_2D CODE CHECK PLS
LOAD<>    D000300 D000320	// LOT 1©ö¢çAU¢¯¡© / L_©öUAU¥ìa 1©ö¢çAU¢¯¡©
AND<>     D000305 D000320	// LOT 1©ö¢çAU¢¯¡© ©öo¨¡U / L_©öUAU¥ìa 1©ö¢çAU¢¯¡©
LOAD<>    D000301 D000321	// LOT 2©ö¢çAU¢¯¡© / L_©öUAU¥ìa 2©ö¢çAU¢¯¡©
AND<>     D000306 D000321	// LOT 2©ö¢çAU¢¯¡© ©öo¨¡U / L_©öUAU¥ìa 2©ö¢çAU¢¯¡©
OR LOAD
LOAD<>    D000302 D000322	// LOT 3©ö¢çAU¢¯¡© / L_©öUAU¥ìa 3©ö¢çAU¢¯¡©
AND<>     D000307 D000322	// LOT 3©ö¢çAU¢¯¡© ©öo¨¡U / L_©öUAU¥ìa 3©ö¢çAU¢¯¡©
OR LOAD
LOAD<>    D000303 D000323	// LOT 4©ö¢çAU¢¯¡© / L_©öUAU¥ìa 4©ö¢çAU¢¯¡©
AND<>     D000308 D000323	// LOT 4©ö¢çAU¢¯¡© ©öo¨¡U / L_©öUAU¥ìa 4©ö¢çAU¢¯¡©
OR LOAD
LOAD<>    D000304 D000324	// LOT 5©ö¢çAU¢¯¡© / L_©öUAU¥ìa 5©ö¢çAU¢¯¡©
AND<>     D000309 D000324	// LOT 5©ö¢çAU¢¯¡© ©öo¨¡U / L_©öUAU¥ìa 5©ö¢çAU¢¯¡©
OR LOAD
AND LOAD
AND NOT   M1902F	// DRY RUN
AND NOT   M19052	// LF_2D CODE SKIP
AND       D003045.1	// 2D 2~5 ©ö©ªA¡Æ ©ö¢çAU¢¯¡© E¢çAI
OUT       M0035F	// LF_2D CODE LOT CODE NG
; L57
LOAD      F00099
BMOV      D007000 D000300 h8008	// LOT NO / LOT 1©ö¢çAU¢¯¡©
BMOV      D007001 D000301 h0008	// LOT 2©ö¢çAU¢¯¡©
BMOV      D007001 D000302 h8008	// LOT 3©ö¢çAU¢¯¡©
BMOV      D007002 D000303 h0008	// LOT 4©ö¢çAU¢¯¡©
BMOV      D007002 D000304 h8008	// LOT 5©ö¢çAU¢¯¡©
; L62
LOAD<=    97 D000300	// LOT 1©ö¢çAU¢¯¡©
SUB       D000300 32 D000305	// LOT 1©ö¢çAU¢¯¡© / LOT 1©ö¢çAU¢¯¡© ©öo¨¡U
; L63
LOAD<=    97 D000301	// LOT 2©ö¢çAU¢¯¡©
SUB       D000301 32 D000306	// LOT 2©ö¢çAU¢¯¡© / LOT 2©ö¢çAU¢¯¡© ©öo¨¡U

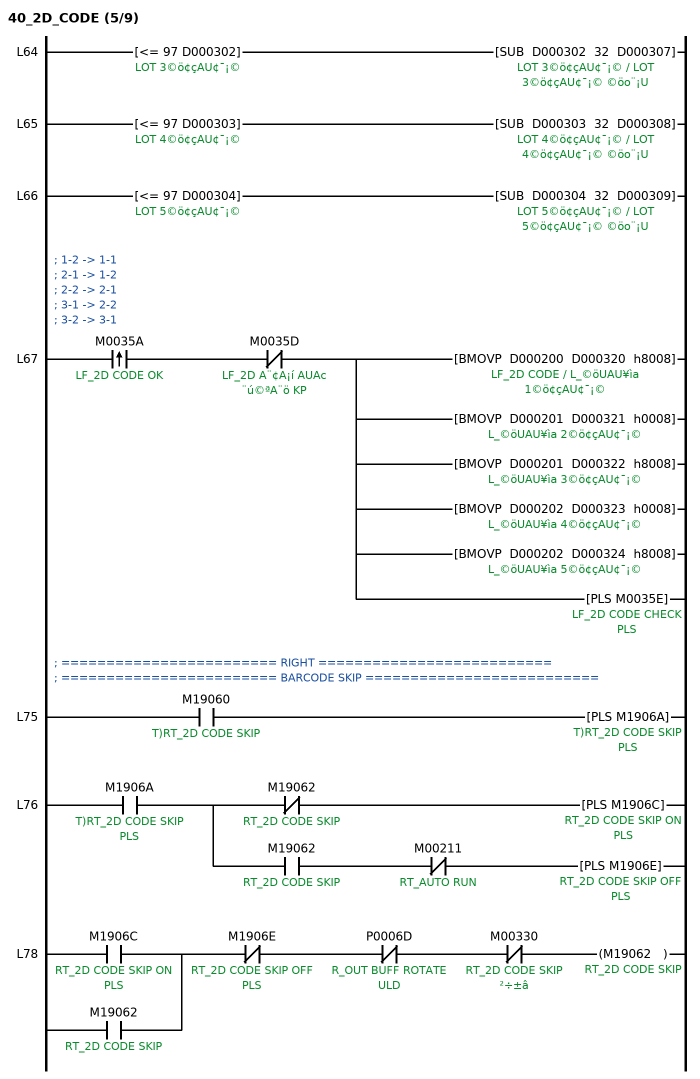
; L64
LOAD<=    97 D000302	// LOT 3©ö¢çAU¢¯¡©
SUB       D000302 32 D000307	// LOT 3©ö¢çAU¢¯¡© / LOT 3©ö¢çAU¢¯¡© ©öo¨¡U
; L65
LOAD<=    97 D000303	// LOT 4©ö¢çAU¢¯¡©
SUB       D000303 32 D000308	// LOT 4©ö¢çAU¢¯¡© / LOT 4©ö¢çAU¢¯¡© ©öo¨¡U
; L66
LOAD<=    97 D000304	// LOT 5©ö¢çAU¢¯¡©
SUB       D000304 32 D000309	// LOT 5©ö¢çAU¢¯¡© / LOT 5©ö¢çAU¢¯¡© ©öo¨¡U
; L67
LOADP     M0035A	// LF_2D CODE OK
AND NOT   M0035D	// LF_2D A¨¢A¡í AUAc ¨ú©ªA¨ö KP
BMOVP     D000200 D000320 h8008	// LF_2D CODE / L_©öUAU¥ìa 1©ö¢çAU¢¯¡©
BMOVP     D000201 D000321 h0008	// L_©öUAU¥ìa 2©ö¢çAU¢¯¡©
BMOVP     D000201 D000322 h8008	// L_©öUAU¥ìa 3©ö¢çAU¢¯¡©
BMOVP     D000202 D000323 h0008	// L_©öUAU¥ìa 4©ö¢çAU¢¯¡©
BMOVP     D000202 D000324 h8008	// L_©öUAU¥ìa 5©ö¢çAU¢¯¡©
OUTP      M0035E	// LF_2D CODE CHECK PLS
// output comment: 1-2 -> 1-1
// output comment: 2-1 -> 1-2
// output comment: 2-2 -> 2-1
// output comment: 3-1 -> 2-2
// output comment: 3-2 -> 3-1
// ======================== RIGHT ==========================
// ======================== BARCODE SKIP ==========================
; L75
LOAD      M19060	// T)RT_2D CODE SKIP
OUTP      M1906A	// T)RT_2D CODE SKIP PLS
; L76
LOAD      M1906A	// T)RT_2D CODE SKIP PLS
MPUSH
AND NOT   M19062	// RT_2D CODE SKIP
OUTP      M1906C	// RT_2D CODE SKIP ON PLS
MPOP
AND       M19062	// RT_2D CODE SKIP
AND NOT   M00211	// RT_AUTO RUN
OUTP      M1906E	// RT_2D CODE SKIP OFF PLS
; L78
LOAD      M1906C	// RT_2D CODE SKIP ON PLS
OR        M19062	// RT_2D CODE SKIP
AND NOT   M1906E	// RT_2D CODE SKIP OFF PLS
AND NOT   P0006D	// R_OUT BUFF ROTATE      ULD
AND NOT   M00330	// RT_2D CODE SKIP ²÷±â
OUT       M19062	// RT_2D CODE SKIP

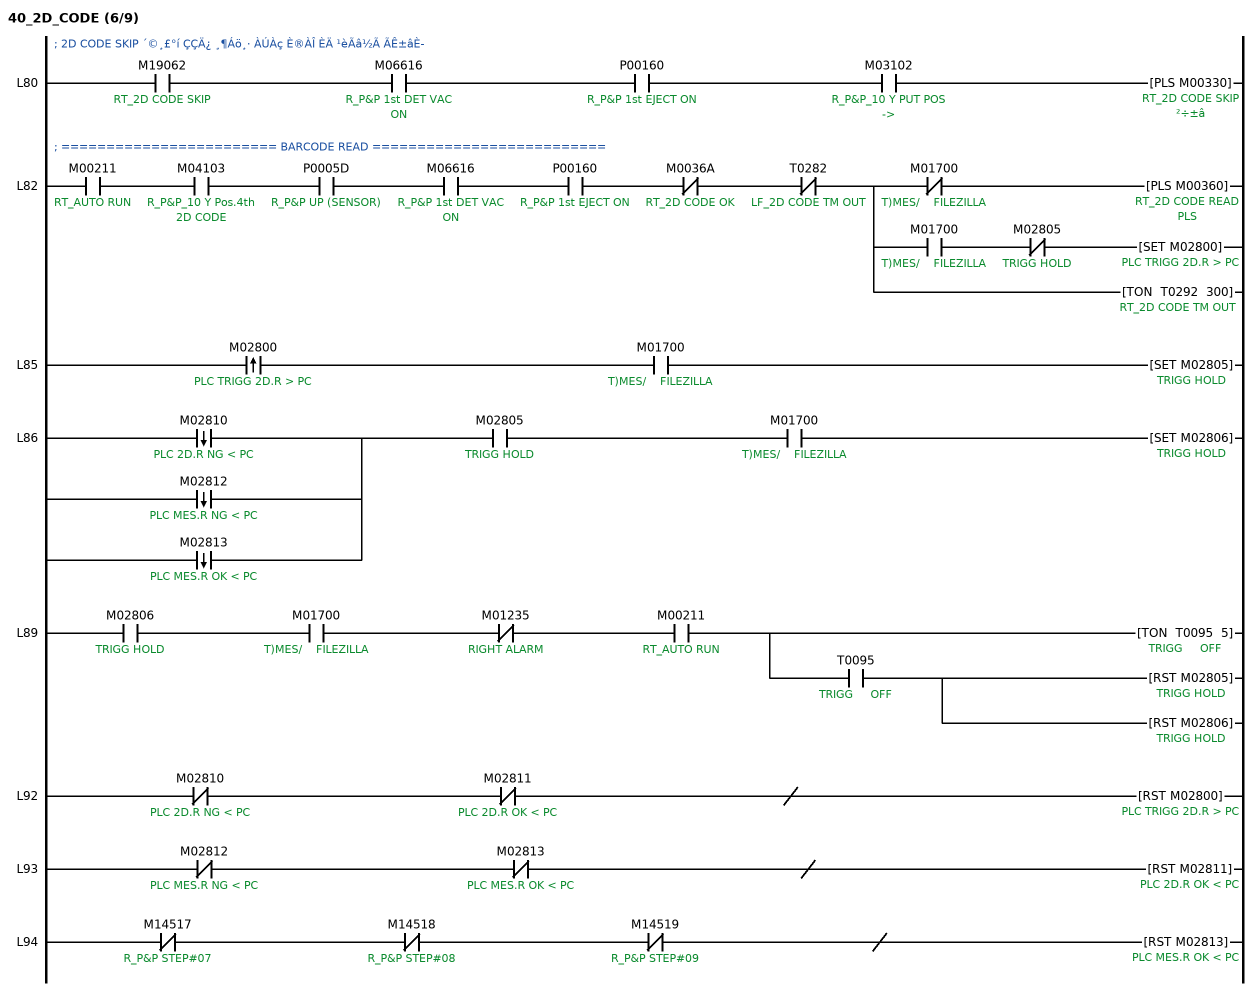
; L80
LOAD      M19062	// RT_2D CODE SKIP
AND       M06616	// R_P&P 1st DET VAC ON
AND       P00160	// R_P&P 1st EJECT ON
AND       M03102	// R_P&P_10 Y PUT POS ->
OUTP      M00330	// RT_2D CODE SKIP ²÷±â
// output comment: 2D CODE SKIP ´©¸£°í ÇÇÄ¿ ¸¶Áö¸· ÀÚÀç È®ÀÎ ÈÄ ¹èÃâ½Ã ÃÊ±âÈ­
// ======================== BARCODE READ ==========================
; L82
LOAD      M00211	// RT_AUTO RUN
AND       M04103	// R_P&P_10 Y Pos.4th 2D CODE
AND       P0005D	// R_P&P UP (SENSOR)
AND       M06616	// R_P&P 1st DET VAC ON
AND       P00160	// R_P&P 1st EJECT ON
AND NOT   M0036A	// RT_2D CODE OK
AND NOT   T0282	// LF_2D CODE TM OUT
MPUSH
AND NOT   M01700	// T)MES/    FILEZILLA
OUTP      M00360	// RT_2D CODE READ PLS
MLOAD
AND       M01700	// T)MES/    FILEZILLA
AND NOT   M02805	// TRIGG HOLD
SET       M02800	// PLC TRIGG 2D.R > PC
MPOP
TON       T0292 300	// RT_2D CODE TM OUT
; L85
LOADP     M02800	// PLC TRIGG 2D.R > PC
AND       M01700	// T)MES/    FILEZILLA
SET       M02805	// TRIGG HOLD
; L86
LOADN     M02810	// PLC 2D.R NG < PC
ORN       M02812	// PLC MES.R NG < PC
ORN       M02813	// PLC MES.R OK < PC
AND       M02805	// TRIGG HOLD
AND       M01700	// T)MES/    FILEZILLA
SET       M02806	// TRIGG HOLD
; L89
LOAD      M02806	// TRIGG HOLD
AND       M01700	// T)MES/    FILEZILLA
AND NOT   M01235	// RIGHT ALARM
AND       M00211	// RT_AUTO RUN
TON       T0095 5	// TRIGG     OFF
AND       T0095	// TRIGG     OFF
RST       M02805	// TRIGG HOLD
RST       M02806	// TRIGG HOLD
; L92
LOAD NOT  M02810	// PLC 2D.R NG < PC
AND NOT   M02811	// PLC 2D.R OK < PC
NOT
RST       M02800	// PLC TRIGG 2D.R > PC
; L93
LOAD NOT  M02812	// PLC MES.R NG < PC
AND NOT   M02813	// PLC MES.R OK < PC
NOT
RST       M02811	// PLC 2D.R OK < PC
; L94
LOAD NOT  M14517	// R_P&P STEP#07
AND NOT   M14518	// R_P&P STEP#08
AND NOT   M14519	// R_P&P STEP#09
NOT
RST       M02813	// PLC MES.R OK < PC

